LIN {X 0,Y 346.568,Z 1182.724,A -85,B 0,C 180,E1 15595.642,E2 15595.642} C_VEL
LIN {X 0,Y 345.198,Z 1187.452,A -85,B 0,C 180,E1 15592.042,E2 15592.042} C_VEL
LIN {X 0,Y 344.384,Z 1191.307,A -85,B 0,C 180,E1 15588.274,E2 15588.274} C_VEL
LIN {X 0,Y 344.008,Z 1194.426,A -85,B 0,C 180,E1 15583.96,E2 15583.96} C_VEL
LIN {X 0,Y 343.921,Z 1195.912,A -85,B 0,C 180,E1 15579.708,E2 15579.708} C_VEL
LIN {X 0,Y 343.92,Z 1196.098,A -85,B 0,C 180,E1 15576.112,E2 15576.112} C_VEL
LIN {X 0,Y 343.929,Z 1195.312,A -85,B 0,C 180,E1 15572.666,E2 15572.666} C_VEL
LIN {X 0,Y 344.029,Z 1193.649,A -85,B 0,C 180,E1 15569.334,E2 15569.334} C_VEL
LIN {X 0,Y 344.332,Z 1190.938,A -85,B 0,C 180,E1 15565.837,E2 15565.837} C_VEL
LIN {X 0,Y 345.025,Z 1187.235,A -85,B 0,C 180,E1 15562.339,E2 15562.339} C_VEL
LIN {X 0,Y 346.225,Z 1182.52,A -85,B 0,C 180,E1 15558.844,E2 15558.844} C_VEL
LIN {X 0,Y 348.076,Z 1176.766,A -85,B 0,C 180,E1 15555.358,E2 15555.358} C_VEL
LIN {X 0,Y 350.938,Z 1169.245,A -85,B 0,C 180,E1 15551.564,E2 15551.564} C_VEL
LIN {X 0,Y 355.746,Z 1158.187,A -85,B 0,C 180,E1 15547.004,E2 15547.004} C_VEL
LIN {X 0,Y 360.656,Z 1147.928,A -85,B 0,C 180,E1 15543.491,E2 15543.491} C_VEL
LIN {X 0,Y 366.084,Z 1137.114,A -85,B 0,C 180,E1 15540.292,E2 15540.292} C_VEL
LIN {X 0,Y 372.756,Z 1124.27,A -85,B 0,C 180,E1 15537.009,E2 15537.009} C_VEL
LIN {X 0,Y 374.75,Z 1120.524,A -85,B 0,C 180,E1 15536.141,E2 15536.141} C_VEL
LIN {X 0,Y 376.046,Z 1116.491,A -85,B 0,C 180,E1 15535.154,E2 15535.154} C_VEL
LIN {X 0,Y 376.596,Z 1106.617,A -85,B 0,C 180,E1 15532.482,E2 15532.482} C_VEL
LIN {X 0,Y 378.202,Z 1102.238,A -85,B 0,C 180,E1 15531.533,E2 15531.533} C_VEL
LIN {X 0,Y 388.069,Z 1083.778,A -85,B 0,C 180,E1 15528.338,E2 15528.338} C_VEL
LIN {X 0,Y 396.837,Z 1066.652,A -85,B 0,C 180,E1 15525.841,E2 15525.841} C_VEL
LIN {X 0,Y 404.683,Z 1050.76,A -85,B 0,C 180,E1 15523.826,E2 15523.826} C_VEL
LIN {X 0,Y 412.691,Z 1033.763,A -85,B 0,C 180,E1 15521.945,E2 15521.945} C_VEL
LIN {X 0,Y 421.387,Z 1014.239,A -85,B 0,C 180,E1 15520.074,E2 15520.074} C_VEL
LIN {X 0,Y 431.348,Z 989.73,A -85,B 0,C 180,E1 15518.098,E2 15518.098} C_VEL
LIN {X 0,Y 438.671,Z 970.006,A -85,B 0,C 180,E1 15516.758,E2 15516.758} C_VEL
LIN {X 0,Y 445.213,Z 950.609,A -85,B 0,C 180,E1 15515.612,E2 15515.612} C_VEL
LIN {X 0,Y 451.627,Z 929.634,A -85,B 0,C 180,E1 15514.556,E2 15514.556} C_VEL
LIN {X 0,Y 458.617,Z 903.499,A -85,B 0,C 180,E1 15513.46,E2 15513.46} C_VEL
LIN {X 0,Y 464.106,Z 878.646,A -85,B 0,C 180,E1 15512.632,E2 15512.632} C_VEL
LIN {X 0,Y 468.081,Z 857.042,A -85,B 0,C 180,E1 15512.046,E2 15512.046} C_VEL
LIN {X 0,Y 471.395,Z 834.774,A -85,B 0,C 180,E1 15511.57,E2 15511.57} C_VEL
LIN {X 0,Y 474.285,Z 806.407,A -85,B 0,C 180,E1 15511.075,E2 15511.075} C_VEL
LIN {X 0,Y 490.886,Z 583.065,A -85,B 0,C 180,E1 15507.599,E2 15507.599} C_VEL
LIN {X 0,Y 493.757,Z 545.15,A -85,B 0,C 180,E1 15507.001,E2 15507.001} C_VEL
LIN {X 0,Y 486.174,Z 532.933,A -85,B 0,C 180,E1 15504.289,E2 15504.289} C_VEL
LIN {X 0,Y 479.89,Z 523.301,A -85,B 0,C 180,E1 15501.699,E2 15501.699} C_VEL
LIN {X 0,Y 474.547,Z 515.365,A -85,B 0,C 180,E1 15499.126,E2 15499.126} C_VEL
LIN {X 0,Y 471.376,Z 510.666,A -85,B 0,C 180,E1 15497.348,E2 15497.348} C_VEL
LIN {X 0,Y 468.645,Z 506.673,A -85,B 0,C 180,E1 15495.595,E2 15495.595} C_VEL
LIN {X 0,Y 465.572,Z 502.135,A -85,B 0,C 180,E1 15493.222,E2 15493.222} C_VEL
LIN {X 0,Y 462.443,Z 497.864,A -85,B 0,C 180,E1 15489.961,E2 15489.961} C_VEL
LIN {X 0,Y 461.806,Z 496.401,A -85,B 0,C 180,E1 15488.969,E2 15488.969} C_VEL
LIN {X 0,Y 459.954,Z 495.059,A -85,B 0,C 180,E1 15483.739,E2 15483.739} C_VEL
LIN {X 0,Y 461.315,Z 496.134,A -85,B 0,C 180,E1 15478.882,E2 15478.882} C_VEL
LIN {X 0,Y 462.041,Z 496.81,A -85,B 0,C 180,E1 15477.768,E2 15477.768} C_VEL
LIN {X 0,Y 464.243,Z 500.766,A -85,B 0,C 180,E1 15475.058,E2 15475.058} C_VEL
LIN {X 0,Y 465.639,Z 502.27,A -85,B 0,C 180,E1 15473.82,E2 15473.82} C_VEL
LIN {X 0,Y 468.799,Z 506.753,A -85,B 0,C 180,E1 15471.414,E2 15471.414} C_VEL
LIN {X 0,Y 473.05,Z 513.167,A -85,B 0,C 180,E1 15468.787,E2 15468.787} C_VEL
LIN {X 0,Y 477.028,Z 519.005,A -85,B 0,C 180,E1 15466.731,E2 15466.731} C_VEL
LIN {X 0,Y 482.506,Z 527.292,A -85,B 0,C 180,E1 15464.279,E2 15464.279} C_VEL
LIN {X 0,Y 489.139,Z 537.554,A -85,B 0,C 180,E1 15461.713,E2 15461.713} C_VEL
LIN {X 0,Y 493.798,Z 546.364,A -85,B 0,C 180,E1 15460.047,E2 15460.047} C_VEL
LIN {X 0,Y 477.206,Z 767.849,A -85,B 0,C 180,E1 15456.603,E2 15456.603} C_VEL
LIN {X 0,Y 472.628,Z 827.074,A -85,B 0,C 180,E1 15455.658,E2 15455.658} C_VEL
LIN {X 0,Y 468.595,Z 857.357,A -85,B 0,C 180,E1 15455.062,E2 15455.062} C_VEL
LIN {X 0,Y 464.454,Z 880.173,A -85,B 0,C 180,E1 15454.482,E2 15454.482} C_VEL
LIN {X 0,Y 459.845,Z 901.491,A -85,B 0,C 180,E1 15453.806,E2 15453.806} C_VEL
LIN {X 0,Y 454.495,Z 922.797,A -85,B 0,C 180,E1 15452.995,E2 15452.995} C_VEL
LIN {X 0,Y 447.013,Z 948.76,A -85,B 0,C 180,E1 15451.797,E2 15451.797} C_VEL
LIN {X 0,Y 439.383,Z 971.659,A -85,B 0,C 180,E1 15450.506,E2 15450.506} C_VEL
LIN {X 0,Y 432.328,Z 990.947,A -85,B 0,C 180,E1 15449.237,E2 15449.237} C_VEL
LIN {X 0,Y 425.139,Z 1009.177,A -85,B 0,C 180,E1 15447.85,E2 15447.85} C_VEL
LIN {X 0,Y 417.318,Z 1027.631,A -85,B 0,C 180,E1 15446.241,E2 15446.241} C_VEL
LIN {X 0,Y 407.206,Z 1049.934,A -85,B 0,C 180,E1 15443.965,E2 15443.965} C_VEL
LIN {X 0,Y 398.127,Z 1068.568,A -85,B 0,C 180,E1 15441.703,E2 15441.703} C_VEL
LIN {X 0,Y 390.292,Z 1084.053,A -85,B 0,C 180,E1 15439.54,E2 15439.54} C_VEL
LIN {X 0,Y 382.689,Z 1098.648,A -85,B 0,C 180,E1 15437.209,E2 15437.209} C_VEL
LIN {X 0,Y 374.954,Z 1113.254,A -85,B 0,C 180,E1 15434.533,E2 15434.533} C_VEL
LIN {X 0,Y 365.691,Z 1130.554,A -85,B 0,C 180,E1 15430.803,E2 15430.803} C_VEL
LIN {X 0,Y 358.982,Z 1143.123,A -85,B 0,C 180,E1 15427.587,E2 15427.587} C_VEL
LIN {X 0,Y 353.255,Z 1154.282,A -85,B 0,C 180,E1 15424.281,E2 15424.281} C_VEL
LIN {X 0,Y 348.218,Z 1164.594,A -85,B 0,C 180,E1 15420.737,E2 15420.737} C_VEL
LIN {X 0,Y 343.21,Z 1175.867,A -85,B 0,C 180,E1 15416.097,E2 15416.097} C_VEL
LIN {X 0,Y 340.131,Z 1183.761,A -85,B 0,C 180,E1 15412.103,E2 15412.103} C_VEL
LIN {X 0,Y 338.181,Z 1189.769,A -85,B 0,C 180,E1 15408.442,E2 15408.442} C_VEL
LIN {X 0,Y 336.997,Z 1194.445,A -85,B 0,C 180,E1 15404.959,E2 15404.959} C_VEL
LIN {X 0,Y 336.305,Z 1198.13,A -85,B 0,C 180,E1 15401.49,E2 15401.49} C_VEL
LIN {X 0,Y 336.02,Z 1200.852,A -85,B 0,C 180,E1 15398.039,E2 15398.039} C_VEL
LIN {X 0,Y 335.924,Z 1202.564,A -85,B 0,C 180,E1 15394.781,E2 15394.781} C_VEL
LIN {X 0,Y 335.915,Z 1203.44,A -85,B 0,C 180,E1 15391.535,E2 15391.535} C_VEL
LIN {X 0,Y 335.913,Z 1203.49,A -85,B 0,C 180,E1 15388.294,E2 15388.294} C_VEL
LIN {X 0,Y 335.926,Z 1202.719,A -85,B 0,C 180,E1 15385.048,E2 15385.048} C_VEL
LIN {X 0,Y 336.037,Z 1201.013,A -85,B 0,C 180,E1 15381.617,E2 15381.617} C_VEL
LIN {X 0,Y 336.388,Z 1198.232,A -85,B 0,C 180,E1 15377.991,E2 15377.991} C_VEL
LIN {X 0,Y 337.167,Z 1194.642,A -85,B 0,C 180,E1 15374.521,E2 15374.521} C_VEL
LIN {X 0,Y 338.55,Z 1189.852,A -85,B 0,C 180,E1 15370.863,E2 15370.863} C_VEL
LIN {X 0,Y 340.701,Z 1183.995,A -85,B 0,C 180,E1 15367.208,E2 15367.208} C_VEL
LIN {X 0,Y 343.862,Z 1176.688,A -85,B 0,C 180,E1 15363.398,E2 15363.398} C_VEL
LIN {X 0,Y 349.185,Z 1166.017,A -85,B 0,C 180,E1 15358.783,E2 15358.783} C_VEL
LIN {X 0,Y 355.02,Z 1155.183,A -85,B 0,C 180,E1 15354.933,E2 15354.933} C_VEL
LIN {X 0,Y 361.14,Z 1144.496,A -85,B 0,C 180,E1 15351.672,E2 15351.672} C_VEL
LIN {X 0,Y 368.243,Z 1132.499,A -85,B 0,C 180,E1 15348.508,E2 15348.508} C_VEL
LIN {X 0,Y 377.138,Z 1117.696,A -85,B 0,C 180,E1 15345.154,E2 15345.154} C_VEL
LIN {X 0,Y 387.584,Z 1099.925,A -85,B 0,C 180,E1 15341.795,E2 15341.795} C_VEL
LIN {X 0,Y 396.6,Z 1084.321,A -85,B 0,C 180,E1 15339.288,E2 15339.288} C_VEL
LIN {X 0,Y 405.359,Z 1068.713,A -85,B 0,C 180,E1 15337.118,E2 15337.118} C_VEL
LIN {X 0,Y 415.508,Z 1049.873,A -85,B 0,C 180,E1 15334.859,E2 15334.859} C_VEL
LIN {X 0,Y 426.712,Z 1027.473,A -85,B 0,C 180,E1 15332.612,E2 15332.612} C_VEL
LIN {X 0,Y 435.312,Z 1009.07,A -85,B 0,C 180,E1 15331.048,E2 15331.048} C_VEL
LIN {X 0,Y 443.198,Z 990.925,A -85,B 0,C 180,E1 15329.708,E2 15329.708} C_VEL
LIN {X 0,Y 450.955,Z 971.577,A -85,B 0,C 180,E1 15328.471,E2 15328.471} C_VEL
LIN {X 0,Y 459.654,Z 947.749,A -85,B 0,C 180,E1 15327.182,E2 15327.182} C_VEL
LIN {X 0,Y 467.531,Z 922.667,A -85,B 0,C 180,E1 15326.077,E2 15326.077} C_VEL
LIN {X 0,Y 473.352,Z 901.443,A -85,B 0,C 180,E1 15325.303,E2 15325.303} C_VEL
LIN {X 0,Y 478.364,Z 880.268,A -85,B 0,C 180,E1 15324.665,E2 15324.665} C_VEL
LIN {X 0,Y 482.642,Z 858.736,A -85,B 0,C 180,E1 15324.14,E2 15324.14} C_VEL
LIN {X 0,Y 486.899,Z 831.241,A -85,B 0,C 180,E1 15323.605,E2 15323.605} C_VEL
LIN {X 0,Y 491.021,Z 786.034,A -85,B 0,C 180,E1 15322.885,E2 15322.885} C_VEL
LIN {X 0,Y 509.816,Z 566.031,A -85,B 0,C 180,E1 15319.504,E2 15319.504} C_VEL
LIN {X 0,Y 510.711,Z 555.321,A -85,B 0,C 180,E1 15319.322,E2 15319.322} C_VEL
LIN {X 0,Y 506.863,Z 548.626,A -85,B 0,C 180,E1 15317.389,E2 15317.389} C_VEL
LIN {X 0,Y 503.453,Z 543.319,A -85,B 0,C 180,E1 15315.434,E2 15315.434} C_VEL
LIN {X 0,Y 501.187,Z 539.639,A -85,B 0,C 180,E1 15313.91,E2 15313.91} C_VEL
LIN {X 0,Y 498.572,Z 535.499,A -85,B 0,C 180,E1 15311.804,E2 15311.804} C_VEL
LIN {X 0,Y 495.748,Z 530.771,A -85,B 0,C 180,E1 15308.584,E2 15308.584} C_VEL
LIN {X 0,Y 493.92,Z 528.892,A -85,B 0,C 180,E1 15303.831,E2 15303.831} C_VEL
LIN {X 0,Y 494.308,Z 529.49,A -85,B 0,C 180,E1 15300.927,E2 15300.927} C_VEL
LIN {X 0,Y 495.953,Z 531.071,A -85,B 0,C 180,E1 15297.92,E2 15297.92} C_VEL
LIN {X 0,Y 498.766,Z 535.705,A -85,B 0,C 180,E1 15294.824,E2 15294.824} C_VEL
LIN {X 0,Y 502.313,Z 541.374,A -85,B 0,C 180,E1 15292.105,E2 15292.105} C_VEL
LIN {X 0,Y 505.598,Z 546.687,A -85,B 0,C 180,E1 15290.093,E2 15290.093} C_VEL
LIN {X 0,Y 509.935,Z 553.595,A -85,B 0,C 180,E1 15287.86,E2 15287.86} C_VEL
LIN {X 0,Y 510.673,Z 555.182,A -85,B 0,C 180,E1 15287.494,E2 15287.494} C_VEL
LIN {X 0,Y 492.196,Z 770.494,A -85,B 0,C 180,E1 15284.188,E2 15284.188} C_VEL
LIN {X 0,Y 487.454,Z 823.866,A -85,B 0,C 180,E1 15283.347,E2 15283.347} C_VEL
LIN {X 0,Y 483.136,Z 853.307,A -85,B 0,C 180,E1 15282.782,E2 15282.782} C_VEL
LIN {X 0,Y 478.728,Z 875.802,A -85,B 0,C 180,E1 15282.224,E2 15282.224} C_VEL
LIN {X 0,Y 473.908,Z 896.408,A -85,B 0,C 180,E1 15281.592,E2 15281.592} C_VEL
LIN {X 0,Y 468.336,Z 916.956,A -85,B 0,C 180,E1 15280.837,E2 15280.837} C_VEL
LIN {X 0,Y 461.23,Z 939.95,A -85,B 0,C 180,E1 15279.827,E2 15279.827} C_VEL
LIN {X 0,Y 452.08,Z 965.513,A -85,B 0,C 180,E1 15278.46,E2 15278.46} C_VEL
LIN {X 0,Y 444.164,Z 985.323,A -85,B 0,C 180,E1 15277.194,E2 15277.194} C_VEL
LIN {X 0,Y 436.186,Z 1003.729,A -85,B 0,C 180,E1 15275.828,E2 15275.828} C_VEL
LIN {X 0,Y 427.778,Z 1021.716,A -85,B 0,C 180,E1 15274.295,E2 15274.295} C_VEL
LIN {X 0,Y 417.178,Z 1043.001,A -85,B 0,C 180,E1 15272.176,E2 15272.176} C_VEL
LIN {X 0,Y 406.533,Z 1062.656,A -85,B 0,C 180,E1 15269.826,E2 15269.826} C_VEL
LIN {X 0,Y 397.526,Z 1078.589,A -85,B 0,C 180,E1 15267.605,E2 15267.605} C_VEL
LIN {X 0,Y 389.142,Z 1092.928,A -85,B 0,C 180,E1 15265.306,E2 15265.306} C_VEL
LIN {X 0,Y 380.303,Z 1107.754,A -85,B 0,C 180,E1 15262.56,E2 15262.56} C_VEL
LIN {X 0,Y 369.726,Z 1125.201,A -85,B 0,C 180,E1 15258.709,E2 15258.709} C_VEL
LIN {X 0,Y 362.319,Z 1137.42,A -85,B 0,C 180,E1 15255.495,E2 15255.495} C_VEL
LIN {X 0,Y 356.234,Z 1147.753,A -85,B 0,C 180,E1 15252.347,E2 15252.347} C_VEL
LIN {X 0,Y 350.658,Z 1157.649,A -85,B 0,C 180,E1 15248.851,E2 15248.851} C_VEL
LIN {X 0,Y 345.045,Z 1168.446,A -85,B 0,C 180,E1 15244.321,E2 15244.321} C_VEL
LIN {X 0,Y 341.235,Z 1176.607,A -85,B 0,C 180,E1 15240.069,E2 15240.069} C_VEL
LIN {X 0,Y 338.869,Z 1182.639,A -85,B 0,C 180,E1 15236.269,E2 15236.269} C_VEL
LIN {X 0,Y 337.392,Z 1187.309,A -85,B 0,C 180,E1 15232.659,E2 15232.659} C_VEL
LIN {X 0,Y 336.513,Z 1190.964,A -85,B 0,C 180,E1 15229.077,E2 15229.077} C_VEL
LIN {X 0,Y 336.103,Z 1193.64,A -85,B 0,C 180,E1 15225.53,E2 15225.53} C_VEL
LIN {X 0,Y 335.947,Z 1195.365,A -85,B 0,C 180,E1 15222.025,E2 15222.025} C_VEL
LIN {X 0,Y 335.919,Z 1196.141,A -85,B 0,C 180,E1 15218.731,E2 15218.731} C_VEL
LIN {X 0,Y 335.92,Z 1196.095,A -85,B 0,C 180,E1 15215.466,E2 15215.466} C_VEL
LIN {X 0,Y 335.935,Z 1195.243,A -85,B 0,C 180,E1 15212.217,E2 15212.217} C_VEL
LIN {X 0,Y 336.05,Z 1193.589,A -85,B 0,C 180,E1 15208.977,E2 15208.977} C_VEL
LIN {X 0,Y 336.367,Z 1190.976,A -85,B 0,C 180,E1 15205.567,E2 15205.567} C_VEL
LIN {X 0,Y 337.119,Z 1187.259,A -85,B 0,C 180,E1 15201.987,E2 15201.987} C_VEL
LIN {X 0,Y 338.413,Z 1182.528,A -85,B 0,C 180,E1 15198.41,E2 15198.41} C_VEL
LIN {X 0,Y 340.488,Z 1176.462,A -85,B 0,C 180,E1 15194.675,E2 15194.675} C_VEL
LIN {X 0,Y 344.061,Z 1167.84,A -85,B 0,C 180,E1 15190.3,E2 15190.3} C_VEL
LIN {X 0,Y 348.939,Z 1157.229,A -85,B 0,C 180,E1 15185.991,E2 15185.991} C_VEL
LIN {X 0,Y 353.92,Z 1147.346,A -85,B 0,C 180,E1 15182.581,E2 15182.581} C_VEL
LIN {X 0,Y 359.513,Z 1136.701,A -85,B 0,C 180,E1 15179.406,E2 15179.406} C_VEL
LIN {X 0,Y 367.403,Z 1122.28,A -85,B 0,C 180,E1 15175.713,E2 15175.713} C_VEL
LIN {X 0,Y 376.061,Z 1106.21,A -85,B 0,C 180,E1 15172.301,E2 15172.301} C_VEL
LIN {X 0,Y 378.202,Z 1102.238,A -85,B 0,C 180,E1 15171.533,E2 15171.533} C_VEL
LIN {X 0,Y 379.88,Z 1097.862,A -85,B 0,C 180,E1 15170.598,E2 15170.598} C_VEL
LIN {X 0,Y 381.583,Z 1086.344,A -85,B 0,C 180,E1 15167.924,E2 15167.924} C_VEL
LIN {X 0,Y 383.266,Z 1082.167,A -85,B 0,C 180,E1 15167.189,E2 15167.189} C_VEL
LIN {X 0,Y 391.871,Z 1065.862,A -85,B 0,C 180,E1 15164.821,E2 15164.821} C_VEL
LIN {X 0,Y 399.975,Z 1049.884,A -85,B 0,C 180,E1 15162.803,E2 15162.803} C_VEL
LIN {X 0,Y 408.506,Z 1032.191,A -85,B 0,C 180,E1 15160.861,E2 15160.861} C_VEL
LIN {X 0,Y 418.945,Z 1009.024,A -85,B 0,C 180,E1 15158.701,E2 15158.701} C_VEL
LIN {X 0,Y 427.583,Z 987.921,A -85,B 0,C 180,E1 15157.053,E2 15157.053} C_VEL
LIN {X 0,Y 434.914,Z 968.488,A -85,B 0,C 180,E1 15155.754,E2 15155.754} C_VEL
LIN {X 0,Y 441.595,Z 948.987,A -85,B 0,C 180,E1 15154.622,E2 15154.622} C_VEL
LIN {X 0,Y 449.208,Z 924.376,A -85,B 0,C 180,E1 15153.417,E2 15153.417} C_VEL
LIN {X 0,Y 455.898,Z 898.52,A -85,B 0,C 180,E1 15152.396,E2 15152.396} C_VEL
LIN {X 0,Y 460.648,Z 877.08,A -85,B 0,C 180,E1 15151.703,E2 15151.703} C_VEL
LIN {X 0,Y 464.647,Z 855.505,A -85,B 0,C 180,E1 15151.133,E2 15151.133} C_VEL
LIN {X 0,Y 468.365,Z 830.302,A -85,B 0,C 180,E1 15150.611,E2 15150.611} C_VEL
LIN {X 0,Y 471.673,Z 793.271,A -85,B 0,C 180,E1 15149.998,E2 15149.998} C_VEL
LIN {X 0,Y 488.775,Z 569.761,A -85,B 0,C 180,E1 15146.528,E2 15146.528} C_VEL
LIN {X 0,Y 490.239,Z 550.028,A -85,B 0,C 180,E1 15146.198,E2 15146.198} C_VEL
LIN {X 0,Y 482.382,Z 537.211,A -85,B 0,C 180,E1 15143.226,E2 15143.226} C_VEL
LIN {X 0,Y 476.274,Z 527.795,A -85,B 0,C 180,E1 15140.524,E2 15140.524} C_VEL
LIN {X 0,Y 470.602,Z 519.114,A -85,B 0,C 180,E1 15137.496,E2 15137.496} C_VEL
LIN {X 0,Y 467.144,Z 514.202,A -85,B 0,C 180,E1 15135.264,E2 15135.264} C_VEL
LIN {X 0,Y 463.967,Z 509.456,A -85,B 0,C 180,E1 15132.699,E2 15132.699} C_VEL
LIN {X 0,Y 461.331,Z 505.676,A -85,B 0,C 180,E1 15129.796,E2 15129.796} C_VEL
LIN {X 0,Y 460.751,Z 504.308,A -85,B 0,C 180,E1 15128.863,E2 15128.863} C_VEL
LIN {X 0,Y 458.978,Z 502.999,A -85,B 0,C 180,E1 15123.747,E2 15123.747} C_VEL
LIN {X 0,Y 460.337,Z 504.081,A -85,B 0,C 180,E1 15118.88,E2 15118.88} C_VEL
LIN {X 0,Y 460.969,Z 504.715,A -85,B 0,C 180,E1 15117.887,E2 15117.887} C_VEL
LIN {X 0,Y 463.132,Z 508.635,A -85,B 0,C 180,E1 15115.17,E2 15115.17} C_VEL
LIN {X 0,Y 464.481,Z 510.181,A -85,B 0,C 180,E1 15113.945,E2 15113.945} C_VEL
LIN {X 0,Y 468.144,Z 515.561,A -85,B 0,C 180,E1 15111.154,E2 15111.154} C_VEL
LIN {X 0,Y 471.623,Z 520.862,A -85,B 0,C 180,E1 15109,E2 15109} C_VEL
LIN {X 0,Y 475.54,Z 526.709,A -85,B 0,C 180,E1 15106.936,E2 15106.936} C_VEL
LIN {X 0,Y 481.28,Z 535.588,A -85,B 0,C 180,E1 15104.331,E2 15104.331} C_VEL
LIN {X 0,Y 487.263,Z 545.065,A -85,B 0,C 180,E1 15101.98,E2 15101.98} C_VEL
LIN {X 0,Y 490.333,Z 551.144,A -85,B 0,C 180,E1 15100.837,E2 15100.837} C_VEL
LIN {X 0,Y 473.346,Z 772.468,A -85,B 0,C 180,E1 15097.4,E2 15097.4} C_VEL
LIN {X 0,Y 468.94,Z 827.656,A -85,B 0,C 180,E1 15096.519,E2 15096.519} C_VEL
LIN {X 0,Y 464.851,Z 857.543,A -85,B 0,C 180,E1 15095.932,E2 15095.932} C_VEL
LIN {X 0,Y 460.661,Z 880.186,A -85,B 0,C 180,E1 15095.359,E2 15095.359} C_VEL
LIN {X 0,Y 456.1,Z 900.89,A -85,B 0,C 180,E1 15094.711,E2 15094.711} C_VEL
LIN {X 0,Y 450.629,Z 922.307,A -85,B 0,C 180,E1 15093.904,E2 15093.904} C_VEL
LIN {X 0,Y 443.158,Z 947.845,A -85,B 0,C 180,E1 15092.74,E2 15092.74} C_VEL
LIN {X 0,Y 435.014,Z 971.75,A -85,B 0,C 180,E1 15091.403,E2 15091.403} C_VEL
LIN {X 0,Y 427.768,Z 991.112,A -85,B 0,C 180,E1 15090.131,E2 15090.131} C_VEL
LIN {X 0,Y 420.123,Z 1009.995,A -85,B 0,C 180,E1 15088.692,E2 15088.692} C_VEL
LIN {X 0,Y 411.515,Z 1029.732,A -85,B 0,C 180,E1 15086.955,E2 15086.955} C_VEL
LIN {X 0,Y 400.691,Z 1052.623,A -85,B 0,C 180,E1 15084.56,E2 15084.56} C_VEL
LIN {X 0,Y 392.15,Z 1069.632,A -85,B 0,C 180,E1 15082.462,E2 15082.462} C_VEL
LIN {X 0,Y 384.07,Z 1085.085,A -85,B 0,C 180,E1 15080.272,E2 15080.272} C_VEL
LIN {X 0,Y 375.661,Z 1100.713,A -85,B 0,C 180,E1 15077.725,E2 15077.725} C_VEL
LIN {X 0,Y 365.605,Z 1118.951,A -85,B 0,C 180,E1 15074.217,E2 15074.217} C_VEL
LIN {X 0,Y 357.76,Z 1132.963,A -85,B 0,C 180,E1 15071.008,E2 15071.008} C_VEL
LIN {X 0,Y 351.354,Z 1144.58,A -85,B 0,C 180,E1 15067.928,E2 15067.928} C_VEL
LIN {X 0,Y 345.498,Z 1155.583,A -85,B 0,C 180,E1 15064.556,E2 15064.556} C_VEL
LIN {X 0,Y 339.274,Z 1167.956,A -85,B 0,C 180,E1 15060.066,E2 15060.066} C_VEL
LIN {X 0,Y 335.072,Z 1177.098,A -85,B 0,C 180,E1 15056.018,E2 15056.018} C_VEL
LIN {X 0,Y 332.214,Z 1184.19,A -85,B 0,C 180,E1 15052.285,E2 15052.285} C_VEL
LIN {X 0,Y 330.208,Z 1190.116,A -85,B 0,C 180,E1 15048.538,E2 15048.538} C_VEL
LIN {X 0,Y 328.903,Z 1195.132,A -85,B 0,C 180,E1 15044.615,E2 15044.615} C_VEL
LIN {X 0,Y 328.15,Z 1199.574,A -85,B 0,C 180,E1 15040.002,E2 15040.002} C_VEL
LIN {X 0,Y 327.942,Z 1202.111,A -85,B 0,C 180,E1 15035.774,E2 15035.774} C_VEL
LIN {X 0,Y 327.913,Z 1203.278,A -85,B 0,C 180,E1 15032.097,E2 15032.097} C_VEL
LIN {X 0,Y 327.916,Z 1203.456,A -85,B 0,C 180,E1 15028.602,E2 15028.602} C_VEL
LIN {X 0,Y 327.928,Z 1202.65,A -85,B 0,C 180,E1 15024.927,E2 15024.927} C_VEL
LIN {X 0,Y 328.05,Z 1200.958,A -85,B 0,C 180,E1 15021.411,E2 15021.411} C_VEL
LIN {X 0,Y 328.437,Z 1198.193,A -85,B 0,C 180,E1 15017.696,E2 15017.696} C_VEL
LIN {X 0,Y 329.332,Z 1194.41,A -85,B 0,C 180,E1 15013.962,E2 15013.962} C_VEL
LIN {X 0,Y 330.853,Z 1189.59,A -85,B 0,C 180,E1 15010.216,E2 15010.216} C_VEL
LIN {X 0,Y 333.193,Z 1183.704,A -85,B 0,C 180,E1 15006.477,E2 15006.477} C_VEL
LIN {X 0,Y 336.785,Z 1176.014,A -85,B 0,C 180,E1 15002.41,E2 15002.41} C_VEL
LIN {X 0,Y 342.779,Z 1164.723,A -85,B 0,C 180,E1 14997.54,E2 14997.54} C_VEL
LIN {X 0,Y 348.791,Z 1154.258,A -85,B 0,C 180,E1 14993.806,E2 14993.806} C_VEL
LIN {X 0,Y 355.32,Z 1143.481,A -85,B 0,C 180,E1 14990.509,E2 14990.509} C_VEL
LIN {X 0,Y 363.201,Z 1130.763,A -85,B 0,C 180,E1 14987.159,E2 14987.159} C_VEL
LIN {X 0,Y 373.952,Z 1113.446,A -85,B 0,C 180,E1 14983.343,E2 14983.343} C_VEL
LIN {X 0,Y 383.086,Z 1098.498,A -85,B 0,C 180,E1 14980.579,E2 14980.579} C_VEL
LIN {X 0,Y 391.943,Z 1083.684,A -85,B 0,C 180,E1 14978.213,E2 14978.213} C_VEL
LIN {X 0,Y 401.418,Z 1067.305,A -85,B 0,C 180,E1 14975.952,E2 14975.952} C_VEL
LIN {X 0,Y 413.3,Z 1045.658,A -85,B 0,C 180,E1 14973.423,E2 14973.423} C_VEL
LIN {X 0,Y 423.336,Z 1025.935,A -85,B 0,C 180,E1 14971.501,E2 14971.501} C_VEL
LIN {X 0,Y 432.189,Z 1007.376,A -85,B 0,C 180,E1 14969.951,E2 14969.951} C_VEL
LIN {X 0,Y 440.294,Z 989.092,A -85,B 0,C 180,E1 14968.632,E2 14968.632} C_VEL
LIN {X 0,Y 449.321,Z 966.871,A -85,B 0,C 180,E1 14967.253,E2 14967.253} C_VEL
LIN {X 0,Y 458.251,Z 941.934,A -85,B 0,C 180,E1 14965.981,E2 14965.981} C_VEL
LIN {X 0,Y 464.824,Z 921.12,A -85,B 0,C 180,E1 14965.097,E2 14965.097} C_VEL
LIN {X 0,Y 470.581,Z 900.399,A -85,B 0,C 180,E1 14964.36,E2 14964.36} C_VEL
LIN {X 0,Y 475.668,Z 879.161,A -85,B 0,C 180,E1 14963.734,E2 14963.734} C_VEL
LIN {X 0,Y 480.278,Z 856.07,A -85,B 0,C 180,E1 14963.186,E2 14963.186} C_VEL
LIN {X 0,Y 484.648,Z 826.198,A -85,B 0,C 180,E1 14962.633,E2 14962.633} C_VEL
LIN {X 0,Y 490.49,Z 760.806,A -85,B 0,C 180,E1 14961.611,E2 14961.611} C_VEL
LIN {X 0,Y 508.048,Z 560.807,A -85,B 0,C 180,E1 14958.548,E2 14958.548} C_VEL
LIN {X 0,Y 504.157,Z 554.3,A -85,B 0,C 180,E1 14956.476,E2 14956.476} C_VEL
LIN {X 0,Y 500.136,Z 547.649,A -85,B 0,C 180,E1 14953.881,E2 14953.881} C_VEL
LIN {X 0,Y 497.344,Z 543.242,A -85,B 0,C 180,E1 14951.598,E2 14951.598} C_VEL
LIN {X 0,Y 494.693,Z 538.674,A -85,B 0,C 180,E1 14948.485,E2 14948.485} C_VEL
LIN {X 0,Y 492.938,Z 536.815,A -85,B 0,C 180,E1 14943.722,E2 14943.722} C_VEL
LIN {X 0,Y 493.368,Z 537.484,A -85,B 0,C 180,E1 14940.813,E2 14940.813} C_VEL
LIN {X 0,Y 494.919,Z 539.073,A -85,B 0,C 180,E1 14937.974,E2 14937.974} C_VEL
LIN {X 0,Y 498.083,Z 544.421,A -85,B 0,C 180,E1 14934.528,E2 14934.528} C_VEL
LIN {X 0,Y 501.058,Z 549.201,A -85,B 0,C 180,E1 14932.259,E2 14932.259} C_VEL
LIN {X 0,Y 504.293,Z 554.533,A -85,B 0,C 180,E1 14930.24,E2 14930.24} C_VEL
LIN {X 0,Y 507.99,Z 560.589,A -85,B 0,C 180,E1 14928.282,E2 14928.282} C_VEL
LIN {X 0,Y 488.97,Z 777.287,A -85,B 0,C 180,E1 14924.97,E2 14924.97} C_VEL
LIN {X 0,Y 484.525,Z 825.48,A -85,B 0,C 180,E1 14924.21,E2 14924.21} C_VEL
LIN {X 0,Y 480.195,Z 853.913,A -85,B 0,C 180,E1 14923.664,E2 14923.664} C_VEL
LIN {X 0,Y 475.748,Z 876.139,A -85,B 0,C 180,E1 14923.118,E2 14923.118} C_VEL
LIN {X 0,Y 470.762,Z 897.009,A -85,B 0,C 180,E1 14922.484,E2 14922.484} C_VEL
LIN {X 0,Y 464.911,Z 918.08,A -85,B 0,C 180,E1 14921.714,E2 14921.714} C_VEL
LIN {X 0,Y 456.877,Z 943.312,A -85,B 0,C 180,E1 14920.6,E2 14920.6} C_VEL
LIN {X 0,Y 448.133,Z 966.801,A -85,B 0,C 180,E1 14919.331,E2 14919.331} C_VEL
LIN {X 0,Y 440.213,Z 986.124,A -85,B 0,C 180,E1 14918.099,E2 14918.099} C_VEL
LIN {X 0,Y 432.403,Z 1003.693,A -85,B 0,C 180,E1 14916.802,E2 14916.802} C_VEL
LIN {X 0,Y 423.777,Z 1021.68,A -85,B 0,C 180,E1 14915.28,E2 14915.28} C_VEL
LIN {X 0,Y 412.889,Z 1042.975,A -85,B 0,C 180,E1 14913.172,E2 14913.172} C_VEL
LIN {X 0,Y 401.853,Z 1062.765,A -85,B 0,C 180,E1 14910.811,E2 14910.811} C_VEL
LIN {X 0,Y 392.514,Z 1078.773,A -85,B 0,C 180,E1 14908.578,E2 14908.578} C_VEL
LIN {X 0,Y 383.374,Z 1093.879,A -85,B 0,C 180,E1 14906.139,E2 14906.139} C_VEL
LIN {X 0,Y 372.766,Z 1111.1,A -85,B 0,C 180,E1 14902.877,E2 14902.877} C_VEL
LIN {X 0,Y 363.202,Z 1126.082,A -85,B 0,C 180,E1 14899.446,E2 14899.446} C_VEL
LIN {X 0,Y 355.635,Z 1138.049,A -85,B 0,C 180,E1 14896.239,E2 14896.239} C_VEL
LIN {X 0,Y 349.146,Z 1148.56,A -85,B 0,C 180,E1 14892.966,E2 14892.966} C_VEL
LIN {X 0,Y 342.572,Z 1159.786,A -85,B 0,C 180,E1 14888.867,E2 14888.867} C_VEL
LIN {X 0,Y 336.981,Z 1169.949,A -85,B 0,C 180,E1 14884.315,E2 14884.315} C_VEL
LIN {X 0,Y 333.494,Z 1177.111,A -85,B 0,C 180,E1 14880.443,E2 14880.443} C_VEL
LIN {X 0,Y 331.103,Z 1182.816,A -85,B 0,C 180,E1 14876.74,E2 14876.74} C_VEL
LIN {X 0,Y 329.523,Z 1187.468,A -85,B 0,C 180,E1 14873.043,E2 14873.043} C_VEL
LIN {X 0,Y 328.571,Z 1191.107,A -85,B 0,C 180,E1 14869.371,E2 14869.371} C_VEL
LIN {X 0,Y 328.113,Z 1193.828,A -85,B 0,C 180,E1 14865.638,E2 14865.638} C_VEL
LIN {X 0,Y 327.946,Z 1195.544,A -85,B 0,C 180,E1 14861.965,E2 14861.965} C_VEL
LIN {X 0,Y 327.916,Z 1196.303,A -85,B 0,C 180,E1 14858.239,E2 14858.239} C_VEL
LIN {X 0,Y 327.917,Z 1196.017,A -85,B 0,C 180,E1 14854.197,E2 14854.197} C_VEL
LIN {X 0,Y 328.017,Z 1194.313,A -85,B 0,C 180,E1 14849.825,E2 14849.825} C_VEL
LIN {X 0,Y 328.34,Z 1191.483,A -85,B 0,C 180,E1 14845.809,E2 14845.809} C_VEL
LIN {X 0,Y 329.125,Z 1187.684,A -85,B 0,C 180,E1 14841.967,E2 14841.967} C_VEL
LIN {X 0,Y 330.452,Z 1183.031,A -85,B 0,C 180,E1 14838.304,E2 14838.304} C_VEL
LIN {X 0,Y 332.478,Z 1177.339,A -85,B 0,C 180,E1 14834.654,E2 14834.654} C_VEL
LIN {X 0,Y 335.465,Z 1170.224,A -85,B 0,C 180,E1 14830.861,E2 14830.861} C_VEL
LIN {X 0,Y 340.242,Z 1160.291,A -85,B 0,C 180,E1 14826.443,E2 14826.443} C_VEL
LIN {X 0,Y 346.205,Z 1148.76,A -85,B 0,C 180,E1 14822.291,E2 14822.291} C_VEL
LIN {X 0,Y 351.929,Z 1138.264,A -85,B 0,C 180,E1 14819.054,E2 14819.054} C_VEL
LIN {X 0,Y 358.542,Z 1126.473,A -85,B 0,C 180,E1 14815.908,E2 14815.908} C_VEL
LIN {X 0,Y 367.399,Z 1110.984,A -85,B 0,C 180,E1 14812.37,E2 14812.37} C_VEL
LIN {X 0,Y 376.873,Z 1093.857,A -85,B 0,C 180,E1 14809.125,E2 14809.125} C_VEL
LIN {X 0,Y 383.266,Z 1082.167,A -85,B 0,C 180,E1 14807.189,E2 14807.189} C_VEL
LIN {X 0,Y 385.174,Z 1077.354,A -85,B 0,C 180,E1 14806.337,E2 14806.337} C_VEL
LIN {X 0,Y 387.469,Z 1065.512,A -85,B 0,C 180,E1 14803.947,E2 14803.947} C_VEL
LIN {X 0,Y 389.584,Z 1060.327,A -85,B 0,C 180,E1 14803.143,E2 14803.143} C_VEL
LIN {X 0,Y 400.455,Z 1038.903,A -85,B 0,C 180,E1 14800.622,E2 14800.622} C_VEL
LIN {X 0,Y 409.201,Z 1020.505,A -85,B 0,C 180,E1 14798.789,E2 14798.789} C_VEL
LIN {X 0,Y 417.074,Z 1002.797,A -85,B 0,C 180,E1 14797.259,E2 14797.259} C_VEL
LIN {X 0,Y 424.873,Z 983.853,A -85,B 0,C 180,E1 14795.834,E2 14795.834} C_VEL
LIN {X 0,Y 433.913,Z 959.888,A -85,B 0,C 180,E1 14794.302,E2 14794.302} C_VEL
LIN {X 0,Y 441.827,Z 935.755,A -85,B 0,C 180,E1 14793.036,E2 14793.036} C_VEL
LIN {X 0,Y 447.808,Z 915.253,A -85,B 0,C 180,E1 14792.131,E2 14792.131} C_VEL
LIN {X 0,Y 452.899,Z 895.386,A -85,B 0,C 180,E1 14791.387,E2 14791.387} C_VEL
LIN {X 0,Y 457.773,Z 873.268,A -85,B 0,C 180,E1 14790.698,E2 14790.698} C_VEL
LIN {X 0,Y 462.739,Z 845.528,A -85,B 0,C 180,E1 14790.021,E2 14790.021} C_VEL
LIN {X 0,Y 465.963,Z 819.816,A -85,B 0,C 180,E1 14789.544,E2 14789.544} C_VEL
LIN {X 0,Y 479.845,Z 643.836,A -85,B 0,C 180,E1 14786.797,E2 14786.797} C_VEL
LIN {X 0,Y 486.897,Z 555.177,A -85,B 0,C 180,E1 14785.417,E2 14785.417} C_VEL
LIN {X 0,Y 480.281,Z 544.19,A -85,B 0,C 180,E1 14782.815,E2 14782.815} C_VEL
LIN {X 0,Y 474.447,Z 535.016,A -85,B 0,C 180,E1 14780.156,E2 14780.156} C_VEL
LIN {X 0,Y 469.124,Z 526.694,A -85,B 0,C 180,E1 14777.233,E2 14777.233} C_VEL
LIN {X 0,Y 465.831,Z 521.916,A -85,B 0,C 180,E1 14775.054,E2 14775.054} C_VEL
LIN {X 0,Y 462.723,Z 517.219,A -85,B 0,C 180,E1 14772.479,E2 14772.479} C_VEL
LIN {X 0,Y 460.184,Z 513.385,A -85,B 0,C 180,E1 14769.568,E2 14769.568} C_VEL
LIN {X 0,Y 459.615,Z 512.169,A -85,B 0,C 180,E1 14768.633,E2 14768.633} C_VEL
LIN {X 0,Y 458,Z 510.937,A -85,B 0,C 180,E1 14763.63,E2 14763.63} C_VEL
LIN {X 0,Y 459.433,Z 512.077,A -85,B 0,C 180,E1 14758.753,E2 14758.753} C_VEL
LIN {X 0,Y 459.935,Z 512.727,A -85,B 0,C 180,E1 14757.944,E2 14757.944} C_VEL
LIN {X 0,Y 462.148,Z 516.641,A -85,B 0,C 180,E1 14755.16,E2 14755.16} C_VEL
LIN {X 0,Y 463.279,Z 517.99,A -85,B 0,C 180,E1 14754.116,E2 14754.116} C_VEL
LIN {X 0,Y 466.875,Z 523.394,A -85,B 0,C 180,E1 14751.316,E2 14751.316} C_VEL
LIN {X 0,Y 470.202,Z 528.555,A -85,B 0,C 180,E1 14749.214,E2 14749.214} C_VEL
LIN {X 0,Y 474.056,Z 534.41,A -85,B 0,C 180,E1 14747.143,E2 14747.143} C_VEL
LIN {X 0,Y 479.851,Z 543.55,A -85,B 0,C 180,E1 14744.469,E2 14744.469} C_VEL
LIN {X 0,Y 485.469,Z 552.716,A -85,B 0,C 180,E1 14742.221,E2 14742.221} C_VEL
LIN {X 0,Y 486.972,Z 555.805,A -85,B 0,C 180,E1 14741.64,E2 14741.64} C_VEL
LIN {X 0,Y 469.631,Z 776.379,A -85,B 0,C 180,E1 14738.222,E2 14738.222} C_VEL
LIN {X 0,Y 465.355,Z 828.269,A -85,B 0,C 180,E1 14737.393,E2 14737.393} C_VEL
LIN {X 0,Y 461.215,Z 857.701,A -85,B 0,C 180,E1 14736.816,E2 14736.816} C_VEL
LIN {X 0,Y 456.981,Z 880.149,A -85,B 0,C 180,E1 14736.253,E2 14736.253} C_VEL
LIN {X 0,Y 452.314,Z 900.924,A -85,B 0,C 180,E1 14735.608,E2 14735.608} C_VEL
LIN {X 0,Y 446.88,Z 921.805,A -85,B 0,C 180,E1 14734.828,E2 14734.828} C_VEL
LIN {X 0,Y 439.428,Z 946.899,A -85,B 0,C 180,E1 14733.7,E2 14733.7} C_VEL
LIN {X 0,Y 430.983,Z 971.219,A -85,B 0,C 180,E1 14732.354,E2 14732.354} C_VEL
LIN {X 0,Y 423.264,Z 991.389,A -85,B 0,C 180,E1 14731.035,E2 14731.035} C_VEL
LIN {X 0,Y 415.52,Z 1010.052,A -85,B 0,C 180,E1 14729.615,E2 14729.615} C_VEL
LIN {X 0,Y 406.165,Z 1030.964,A -85,B 0,C 180,E1 14727.771,E2 14727.771} C_VEL
LIN {X 0,Y 395.582,Z 1052.648,A -85,B 0,C 180,E1 14725.485,E2 14725.485} C_VEL
LIN {X 0,Y 387.068,Z 1069.132,A -85,B 0,C 180,E1 14723.452,E2 14723.452} C_VEL
LIN {X 0,Y 378.768,Z 1084.535,A -85,B 0,C 180,E1 14721.27,E2 14721.27} C_VEL
LIN {X 0,Y 370.301,Z 1099.759,A -85,B 0,C 180,E1 14718.787,E2 14718.787} C_VEL
LIN {X 0,Y 360.458,Z 1117.155,A -85,B 0,C 180,E1 14715.469,E2 14715.469} C_VEL
LIN {X 0,Y 351.507,Z 1132.488,A -85,B 0,C 180,E1 14711.948,E2 14711.948} C_VEL
LIN {X 0,Y 344.722,Z 1144.272,A -85,B 0,C 180,E1 14708.792,E2 14708.792} C_VEL
LIN {X 0,Y 338.571,Z 1155.302,A -85,B 0,C 180,E1 14705.368,E2 14705.368} C_VEL
LIN {X 0,Y 332.188,Z 1167.414,A -85,B 0,C 180,E1 14700.923,E2 14700.923} C_VEL
LIN {X 0,Y 327.578,Z 1176.885,A -85,B 0,C 180,E1 14696.659,E2 14696.659} C_VEL
LIN {X 0,Y 324.539,Z 1183.995,A -85,B 0,C 180,E1 14692.842,E2 14692.842} C_VEL
LIN {X 0,Y 322.476,Z 1189.682,A -85,B 0,C 180,E1 14689.187,E2 14689.187} C_VEL
LIN {X 0,Y 321.089,Z 1194.556,A -85,B 0,C 180,E1 14685.348,E2 14685.348} C_VEL
LIN {X 0,Y 320.285,Z 1198.503,A -85,B 0,C 180,E1 14681.342,E2 14681.342} C_VEL
LIN {X 0,Y 319.966,Z 1201.642,A -85,B 0,C 180,E1 14676.82,E2 14676.82} C_VEL
LIN {X 0,Y 319.915,Z 1203.137,A -85,B 0,C 180,E1 14672.508,E2 14672.508} C_VEL
LIN {X 0,Y 319.916,Z 1203.398,A -85,B 0,C 180,E1 14668.746,E2 14668.746} C_VEL
LIN {X 0,Y 319.927,Z 1202.653,A -85,B 0,C 180,E1 14664.98,E2 14664.98} C_VEL
LIN {X 0,Y 320.064,Z 1200.905,A -85,B 0,C 180,E1 14661.195,E2 14661.195} C_VEL
LIN {X 0,Y 320.49,Z 1198.154,A -85,B 0,C 180,E1 14657.386,E2 14657.386} C_VEL
LIN {X 0,Y 321.458,Z 1194.388,A -85,B 0,C 180,E1 14653.558,E2 14653.558} C_VEL
LIN {X 0,Y 323.137,Z 1189.486,A -85,B 0,C 180,E1 14649.65,E2 14649.65} C_VEL
LIN {X 0,Y 325.707,Z 1183.478,A -85,B 0,C 180,E1 14645.751,E2 14645.751} C_VEL
LIN {X 0,Y 329.801,Z 1175.344,A -85,B 0,C 180,E1 14641.379,E2 14641.379} C_VEL
LIN {X 0,Y 335.988,Z 1164.343,A -85,B 0,C 180,E1 14636.596,E2 14636.596} C_VEL
LIN {X 0,Y 342.195,Z 1154.161,A -85,B 0,C 180,E1 14632.912,E2 14632.912} C_VEL
LIN {X 0,Y 348.894,Z 1143.608,A -85,B 0,C 180,E1 14629.634,E2 14629.634} C_VEL
LIN {X 0,Y 356.687,Z 1131.546,A -85,B 0,C 180,E1 14626.403,E2 14626.403} C_VEL
LIN {X 0,Y 367.336,Z 1115.179,A -85,B 0,C 180,E1 14622.7,E2 14622.7} C_VEL
LIN {X 0,Y 377.738,Z 1098.742,A -85,B 0,C 180,E1 14619.622,E2 14619.622} C_VEL
LIN {X 0,Y 387.17,Z 1083.491,A -85,B 0,C 180,E1 14617.18,E2 14617.18} C_VEL
LIN {X 0,Y 397.23,Z 1066.628,A -85,B 0,C 180,E1 14614.859,E2 14614.859} C_VEL
LIN {X 0,Y 409.627,Z 1044.584,A -85,B 0,C 180,E1 14612.315,E2 14612.315} C_VEL
LIN {X 0,Y 419.274,Z 1026.127,A -85,B 0,C 180,E1 14610.529,E2 14610.529} C_VEL
LIN {X 0,Y 428.022,Z 1008.265,A -85,B 0,C 180,E1 14609.04,E2 14609.04} C_VEL
LIN {X 0,Y 436.368,Z 989.936,A -85,B 0,C 180,E1 14607.72,E2 14607.72} C_VEL
LIN {X 0,Y 444.618,Z 970.179,A -85,B 0,C 180,E1 14606.489,E2 14606.489} C_VEL
LIN {X 0,Y 454.083,Z 944.998,A -85,B 0,C 180,E1 14605.178,E2 14605.178} C_VEL
LIN {X 0,Y 461.724,Z 921.371,A -85,B 0,C 180,E1 14604.176,E2 14604.176} C_VEL
LIN {X 0,Y 467.561,Z 900.804,A -85,B 0,C 180,E1 14603.452,E2 14603.452} C_VEL
LIN {X 0,Y 472.713,Z 879.766,A -85,B 0,C 180,E1 14602.838,E2 14602.838} C_VEL
LIN {X 0,Y 477.217,Z 857.793,A -85,B 0,C 180,E1 14602.318,E2 14602.318} C_VEL
LIN {X 0,Y 481.672,Z 829.257,A -85,B 0,C 180,E1 14601.783,E2 14601.783} C_VEL
LIN {X 0,Y 486.182,Z 781.402,A -85,B 0,C 180,E1 14601.032,E2 14601.032} C_VEL
LIN {X 0,Y 505.44,Z 566.529,A -85,B 0,C 180,E1 14597.761,E2 14597.761} C_VEL
LIN {X 0,Y 501.406,Z 559.654,A -85,B 0,C 180,E1 14595.44,E2 14595.44} C_VEL
LIN {X 0,Y 498.531,Z 554.952,A -85,B 0,C 180,E1 14593.454,E2 14593.454} C_VEL
LIN {X 0,Y 496.121,Z 550.984,A -85,B 0,C 180,E1 14591.391,E2 14591.391} C_VEL
LIN {X 0,Y 493.64,Z 546.577,A -85,B 0,C 180,E1 14588.386,E2 14588.386} C_VEL
LIN {X 0,Y 491.96,Z 544.755,A -85,B 0,C 180,E1 14583.711,E2 14583.711} C_VEL
LIN {X 0,Y 492.429,Z 545.478,A -85,B 0,C 180,E1 14580.698,E2 14580.698} C_VEL
LIN {X 0,Y 493.85,Z 546.966,A -85,B 0,C 180,E1 14578.086,E2 14578.086} C_VEL
LIN {X 0,Y 496.893,Z 552.221,A -85,B 0,C 180,E1 14574.689,E2 14574.689} C_VEL
LIN {X 0,Y 499.729,Z 556.877,A -85,B 0,C 180,E1 14572.469,E2 14572.469} C_VEL
LIN {X 0,Y 502.897,Z 562.215,A -85,B 0,C 180,E1 14570.443,E2 14570.443} C_VEL
LIN {X 0,Y 505.358,Z 566.495,A -85,B 0,C 180,E1 14569.071,E2 14569.071} C_VEL
LIN {X 0,Y 486.056,Z 781.6,A -85,B 0,C 180,E1 14565.8,E2 14565.8} C_VEL
LIN {X 0,Y 481.723,Z 827.025,A -85,B 0,C 180,E1 14565.085,E2 14565.085} C_VEL
LIN {X 0,Y 477.366,Z 854.555,A -85,B 0,C 180,E1 14564.556,E2 14564.556} C_VEL
LIN {X 0,Y 472.887,Z 876.482,A -85,B 0,C 180,E1 14564.023,E2 14564.023} C_VEL
LIN {X 0,Y 467.711,Z 897.686,A -85,B 0,C 180,E1 14563.386,E2 14563.386} C_VEL
LIN {X 0,Y 461.621,Z 919.127,A -85,B 0,C 180,E1 14562.608,E2 14562.608} C_VEL
LIN {X 0,Y 452.981,Z 945.348,A -85,B 0,C 180,E1 14561.447,E2 14561.447} C_VEL
LIN {X 0,Y 444.57,Z 967.414,A -85,B 0,C 180,E1 14560.258,E2 14560.258} C_VEL
LIN {X 0,Y 436.374,Z 986.926,A -85,B 0,C 180,E1 14559.019,E2 14559.019} C_VEL
LIN {X 0,Y 428.389,Z 1004.423,A -85,B 0,C 180,E1 14557.733,E2 14557.733} C_VEL
LIN {X 0,Y 419.219,Z 1023.037,A -85,B 0,C 180,E1 14556.158,E2 14556.158} C_VEL
LIN {X 0,Y 407.08,Z 1045.85,A -85,B 0,C 180,E1 14553.861,E2 14553.861} C_VEL
LIN {X 0,Y 396.903,Z 1063.55,A -85,B 0,C 180,E1 14551.731,E2 14551.731} C_VEL
LIN {X 0,Y 387.45,Z 1079.24,A -85,B 0,C 180,E1 14549.533,E2 14549.533} C_VEL
LIN {X 0,Y 378.077,Z 1094.218,A -85,B 0,C 180,E1 14547.104,E2 14547.104} C_VEL
LIN {X 0,Y 367.397,Z 1110.918,A -85,B 0,C 180,E1 14543.927,E2 14543.927} C_VEL
LIN {X 0,Y 357.016,Z 1126.555,A -85,B 0,C 180,E1 14540.315,E2 14540.315} C_VEL
LIN {X 0,Y 349.274,Z 1138.291,A -85,B 0,C 180,E1 14537.125,E2 14537.125} C_VEL
LIN {X 0,Y 342.435,Z 1148.842,A -85,B 0,C 180,E1 14533.789,E2 14533.789} C_VEL
LIN {X 0,Y 335.237,Z 1160.553,A -85,B 0,C 180,E1 14529.42,E2 14529.42} C_VEL
LIN {X 0,Y 329.413,Z 1170.527,A -85,B 0,C 180,E1 14524.794,E2 14524.794} C_VEL
LIN {X 0,Y 325.764,Z 1177.617,A -85,B 0,C 180,E1 14520.835,E2 14520.835} C_VEL
LIN {X 0,Y 323.157,Z 1183.511,A -85,B 0,C 180,E1 14516.855,E2 14516.855} C_VEL
LIN {X 0,Y 321.291,Z 1188.884,A -85,B 0,C 180,E1 14512.313,E2 14512.313} C_VEL
LIN {X 0,Y 320.296,Z 1192.982,A -85,B 0,C 180,E1 14507.438,E2 14507.438} C_VEL
LIN {X 0,Y 319.997,Z 1195.113,A -85,B 0,C 180,E1 14503.553,E2 14503.553} C_VEL
LIN {X 0,Y 319.925,Z 1196.198,A -85,B 0,C 180,E1 14499.898,E2 14499.898} C_VEL
LIN {X 0,Y 319.92,Z 1196.37,A -85,B 0,C 180,E1 14496.28,E2 14496.28} C_VEL
LIN {X 0,Y 319.931,Z 1195.643,A -85,B 0,C 180,E1 14492.687,E2 14492.687} C_VEL
LIN {X 0,Y 320.057,Z 1193.913,A -85,B 0,C 180,E1 14488.926,E2 14488.926} C_VEL
LIN {X 0,Y 320.401,Z 1191.361,A -85,B 0,C 180,E1 14485.346,E2 14485.346} C_VEL
LIN {X 0,Y 321.226,Z 1187.704,A -85,B 0,C 180,E1 14481.588,E2 14481.588} C_VEL
LIN {X 0,Y 322.653,Z 1183.034,A -85,B 0,C 180,E1 14477.835,E2 14477.835} C_VEL
LIN {X 0,Y 324.82,Z 1177.325,A -85,B 0,C 180,E1 14474.1,E2 14474.1} C_VEL
LIN {X 0,Y 327.993,Z 1170.194,A -85,B 0,C 180,E1 14470.222,E2 14470.222} C_VEL
LIN {X 0,Y 333.047,Z 1160.222,A -85,B 0,C 180,E1 14465.714,E2 14465.714} C_VEL
LIN {X 0,Y 339.304,Z 1148.67,A -85,B 0,C 180,E1 14461.486,E2 14461.486} C_VEL
LIN {X 0,Y 345.31,Z 1138.149,A -85,B 0,C 180,E1 14458.198,E2 14458.198} C_VEL
LIN {X 0,Y 351.854,Z 1126.95,A -85,B 0,C 180,E1 14455.168,E2 14455.168} C_VEL
LIN {X 0,Y 360.032,Z 1113.104,A -85,B 0,C 180,E1 14451.937,E2 14451.937} C_VEL
LIN {X 0,Y 370.493,Z 1094.996,A -85,B 0,C 180,E1 14448.403,E2 14448.403} C_VEL
LIN {X 0,Y 379.109,Z 1079.654,A -85,B 0,C 180,E1 14445.872,E2 14445.872} C_VEL
LIN {X 0,Y 387.297,Z 1064.574,A -85,B 0,C 180,E1 14443.709,E2 14443.709} C_VEL
LIN {X 0,Y 389.584,Z 1060.327,A -85,B 0,C 180,E1 14443.143,E2 14443.143} C_VEL
LIN {X 0,Y 391.732,Z 1055.133,A -85,B 0,C 180,E1 14442.356,E2 14442.356} C_VEL
LIN {X 0,Y 394.821,Z 1041.552,A -85,B 0,C 180,E1 14440.025,E2 14440.025} C_VEL
LIN {X 0,Y 396.756,Z 1036.692,A -85,B 0,C 180,E1 14439.422,E2 14439.422} C_VEL
LIN {X 0,Y 404.999,Z 1019.721,A -85,B 0,C 180,E1 14437.755,E2 14437.755} C_VEL
LIN {X 0,Y 412.931,Z 1002.284,A -85,B 0,C 180,E1 14436.263,E2 14436.263} C_VEL
LIN {X 0,Y 421.254,Z 982.482,A -85,B 0,C 180,E1 14434.791,E2 14434.791} C_VEL
LIN {X 0,Y 431.163,Z 956.205,A -85,B 0,C 180,E1 14433.16,E2 14433.16} C_VEL
LIN {X 0,Y 438.195,Z 935.087,A -85,B 0,C 180,E1 14432.075,E2 14432.075} C_VEL
LIN {X 0,Y 444.176,Z 914.937,A -85,B 0,C 180,E1 14431.197,E2 14431.197} C_VEL
LIN {X 0,Y 449.524,Z 894.366,A -85,B 0,C 180,E1 14430.437,E2 14430.437} C_VEL
LIN {X 0,Y 454.834,Z 870.487,A -85,B 0,C 180,E1 14429.712,E2 14429.712} C_VEL
LIN {X 0,Y 459.806,Z 841.826,A -85,B 0,C 180,E1 14429.047,E2 14429.047} C_VEL
LIN {X 0,Y 462.686,Z 818.651,A -85,B 0,C 180,E1 14428.626,E2 14428.626} C_VEL
LIN {X 0,Y 479.238,Z 613.765,A -85,B 0,C 180,E1 14425.443,E2 14425.443} C_VEL
LIN {X 0,Y 483.63,Z 560.286,A -85,B 0,C 180,E1 14424.62,E2 14424.62} C_VEL
LIN {X 0,Y 477.8,Z 550.542,A -85,B 0,C 180,E1 14422.226,E2 14422.226} C_VEL
LIN {X 0,Y 472.52,Z 542.058,A -85,B 0,C 180,E1 14419.726,E2 14419.726} C_VEL
LIN {X 0,Y 467.655,Z 534.272,A -85,B 0,C 180,E1 14416.969,E2 14416.969} C_VEL
LIN {X 0,Y 464.523,Z 529.63,A -85,B 0,C 180,E1 14414.842,E2 14414.842} C_VEL
LIN {X 0,Y 461.486,Z 524.98,A -85,B 0,C 180,E1 14412.259,E2 14412.259} C_VEL
LIN {X 0,Y 459.007,Z 520.99,A -85,B 0,C 180,E1 14409.277,E2 14409.277} C_VEL
LIN {X 0,Y 458.566,Z 520.075,A -85,B 0,C 180,E1 14408.527,E2 14408.527} C_VEL
LIN {X 0,Y 457.024,Z 518.874,A -85,B 0,C 180,E1 14403.512,E2 14403.512} C_VEL
LIN {X 0,Y 458.612,Z 520.119,A -85,B 0,C 180,E1 14398.501,E2 14398.501} C_VEL
LIN {X 0,Y 461.295,Z 524.77,A -85,B 0,C 180,E1 14395.026,E2 14395.026} C_VEL
LIN {X 0,Y 462.145,Z 525.929,A -85,B 0,C 180,E1 14394.226,E2 14394.226} C_VEL
LIN {X 0,Y 465.527,Z 531.073,A -85,B 0,C 180,E1 14391.539,E2 14391.539} C_VEL
LIN {X 0,Y 468.788,Z 536.244,A -85,B 0,C 180,E1 14389.43,E2 14389.43} C_VEL
LIN {X 0,Y 472.812,Z 542.456,A -85,B 0,C 180,E1 14387.233,E2 14387.233} C_VEL
LIN {X 0,Y 478.967,Z 552.357,A -85,B 0,C 180,E1 14384.377,E2 14384.377} C_VEL
LIN {X 0,Y 483.703,Z 560.469,A -85,B 0,C 180,E1 14382.453,E2 14382.453} C_VEL
LIN {X 0,Y 466.017,Z 780.198,A -85,B 0,C 180,E1 14379.058,E2 14379.058} C_VEL
LIN {X 0,Y 461.872,Z 828.95,A -85,B 0,C 180,E1 14378.279,E2 14378.279} C_VEL
LIN {X 0,Y 457.691,Z 857.86,A -85,B 0,C 180,E1 14377.713,E2 14377.713} C_VEL
LIN {X 0,Y 453.42,Z 880.086,A -85,B 0,C 180,E1 14377.161,E2 14377.161} C_VEL
LIN {X 0,Y 448.566,Z 901.252,A -85,B 0,C 180,E1 14376.509,E2 14376.509} C_VEL
LIN {X 0,Y 442.699,Z 923.26,A -85,B 0,C 180,E1 14375.689,E2 14375.689} C_VEL
LIN {X 0,Y 434.381,Z 950.095,A -85,B 0,C 180,E1 14374.462,E2 14374.462} C_VEL
LIN {X 0,Y 426.607,Z 971.916,A -85,B 0,C 180,E1 14373.248,E2 14373.248} C_VEL
LIN {X 0,Y 419.041,Z 991.246,A -85,B 0,C 180,E1 14371.987,E2 14371.987} C_VEL
LIN {X 0,Y 411.354,Z 1009.351,A -85,B 0,C 180,E1 14370.62,E2 14370.62} C_VEL
LIN {X 0,Y 402.291,Z 1029.136,A -85,B 0,C 180,E1 14368.895,E2 14368.895} C_VEL
LIN {X 0,Y 390.877,Z 1052.105,A -85,B 0,C 180,E1 14366.501,E2 14366.501} C_VEL
LIN {X 0,Y 381.818,Z 1069.146,A -85,B 0,C 180,E1 14364.399,E2 14364.399} C_VEL
LIN {X 0,Y 373.255,Z 1084.562,A -85,B 0,C 180,E1 14362.207,E2 14362.207} C_VEL
LIN {X 0,Y 364.474,Z 1099.857,A -85,B 0,C 180,E1 14359.697,E2 14359.697} C_VEL
LIN {X 0,Y 354.12,Z 1117.502,A -85,B 0,C 180,E1 14356.287,E2 14356.287} C_VEL
LIN {X 0,Y 345.264,Z 1132.15,A -85,B 0,C 180,E1 14352.886,E2 14352.886} C_VEL
LIN {X 0,Y 338.18,Z 1143.962,A -85,B 0,C 180,E1 14349.689,E2 14349.689} C_VEL
LIN {X 0,Y 331.714,Z 1155.015,A -85,B 0,C 180,E1 14346.213,E2 14346.213} C_VEL
LIN {X 0,Y 325.071,Z 1167.064,A -85,B 0,C 180,E1 14341.733,E2 14341.733} C_VEL
LIN {X 0,Y 320.122,Z 1176.666,A -85,B 0,C 180,E1 14337.331,E2 14337.331} C_VEL
LIN {X 0,Y 316.895,Z 1183.799,A -85,B 0,C 180,E1 14333.425,E2 14333.425} C_VEL
LIN {X 0,Y 314.684,Z 1189.505,A -85,B 0,C 180,E1 14329.682,E2 14329.682} C_VEL
LIN {X 0,Y 313.191,Z 1194.396,A -85,B 0,C 180,E1 14325.745,E2 14325.745} C_VEL
LIN {X 0,Y 312.344,Z 1198.199,A -85,B 0,C 180,E1 14321.822,E2 14321.822} C_VEL
LIN {X 0,Y 312.002,Z 1201.059,A -85,B 0,C 180,E1 14317.735,E2 14317.735} C_VEL
LIN {X 0,Y 311.917,Z 1202.926,A -85,B 0,C 180,E1 14313.308,E2 14313.308} C_VEL
LIN {X 0,Y 311.914,Z 1203.341,A -85,B 0,C 180,E1 14308.898,E2 14308.898} C_VEL
LIN {X 0,Y 311.929,Z 1202.586,A -85,B 0,C 180,E1 14304.851,E2 14304.851} C_VEL
LIN {X 0,Y 312.077,Z 1200.854,A -85,B 0,C 180,E1 14300.968,E2 14300.968} C_VEL
LIN {X 0,Y 312.547,Z 1198.118,A -85,B 0,C 180,E1 14297.06,E2 14297.06} C_VEL
LIN {X 0,Y 313.596,Z 1194.367,A -85,B 0,C 180,E1 14293.134,E2 14293.134} C_VEL
LIN {X 0,Y 315.364,Z 1189.582,A -85,B 0,C 180,E1 14289.201,E2 14289.201} C_VEL
LIN {X 0,Y 318.023,Z 1183.734,A -85,B 0,C 180,E1 14285.282,E2 14285.282} C_VEL
LIN {X 0,Y 321.877,Z 1176.437,A -85,B 0,C 180,E1 14281.218,E2 14281.218} C_VEL
LIN {X 0,Y 328.217,Z 1165.79,A -85,B 0,C 180,E1 14276.328,E2 14276.328} C_VEL
LIN {X 0,Y 335.423,Z 1154.463,A -85,B 0,C 180,E1 14272.116,E2 14272.116} C_VEL
LIN {X 0,Y 342.544,Z 1143.738,A -85,B 0,C 180,E1 14268.725,E2 14268.725} C_VEL
LIN {X 0,Y 350.667,Z 1131.703,A -85,B 0,C 180,E1 14265.459,E2 14265.459} C_VEL
LIN {X 0,Y 361.736,Z 1115.395,A -85,B 0,C 180,E1 14261.73,E2 14261.73} C_VEL
LIN {X 0,Y 372.502,Z 1098.992,A -85,B 0,C 180,E1 14258.639,E2 14258.639} C_VEL
LIN {X 0,Y 381.933,Z 1084.25,A -85,B 0,C 180,E1 14256.263,E2 14256.263} C_VEL
LIN {X 0,Y 391.666,Z 1068.446,A -85,B 0,C 180,E1 14254.066,E2 14254.066} C_VEL
LIN {X 0,Y 403.413,Z 1048.468,A -85,B 0,C 180,E1 14251.699,E2 14251.699} C_VEL
LIN {X 0,Y 415.062,Z 1026.856,A -85,B 0,C 180,E1 14249.585,E2 14249.585} C_VEL
LIN {X 0,Y 424.307,Z 1008.448,A -85,B 0,C 180,E1 14248.056,E2 14248.056} C_VEL
LIN {X 0,Y 432.915,Z 989.995,A -85,B 0,C 180,E1 14246.74,E2 14246.74} C_VEL
LIN {X 0,Y 441.096,Z 970.84,A -85,B 0,C 180,E1 14245.556,E2 14245.556} C_VEL
LIN {X 0,Y 450.374,Z 946.911,A -85,B 0,C 180,E1 14244.31,E2 14244.31} C_VEL
LIN {X 0,Y 458.69,Z 921.819,A -85,B 0,C 180,E1 14243.25,E2 14243.25} C_VEL
LIN {X 0,Y 464.832,Z 900.595,A -85,B 0,C 180,E1 14242.513,E2 14242.513} C_VEL
LIN {X 0,Y 470.024,Z 879.754,A -85,B 0,C 180,E1 14241.914,E2 14241.914} C_VEL
LIN {X 0,Y 474.603,Z 857.793,A -85,B 0,C 180,E1 14241.403,E2 14241.403} C_VEL
LIN {X 0,Y 479.122,Z 829.416,A -85,B 0,C 180,E1 14240.876,E2 14240.876} C_VEL
LIN {X 0,Y 483.711,Z 781.863,A -85,B 0,C 180,E1 14240.134,E2 14240.134} C_VEL
LIN {X 0,Y 502.915,Z 572.266,A -85,B 0,C 180,E1 14236.96,E2 14236.96} C_VEL
LIN {X 0,Y 499.453,Z 566.425,A -85,B 0,C 180,E1 14234.848,E2 14234.848} C_VEL
LIN {X 0,Y 497.178,Z 562.553,A -85,B 0,C 180,E1 14233.195,E2 14233.195} C_VEL
LIN {X 0,Y 495.027,Z 558.871,A -85,B 0,C 180,E1 14231.299,E2 14231.299} C_VEL
LIN {X 0,Y 492.509,Z 554.427,A -85,B 0,C 180,E1 14228.17,E2 14228.17} C_VEL
LIN {X 0,Y 490.981,Z 552.68,A -85,B 0,C 180,E1 14223.62,E2 14223.62} C_VEL
LIN {X 0,Y 491.493,Z 553.475,A -85,B 0,C 180,E1 14220.583,E2 14220.583} C_VEL
LIN {X 0,Y 492.784,Z 554.857,A -85,B 0,C 180,E1 14218.198,E2 14218.198} C_VEL
LIN {X 0,Y 495.706,Z 560.019,A -85,B 0,C 180,E1 14214.85,E2 14214.85} C_VEL
LIN {X 0,Y 498.484,Z 564.7,A -85,B 0,C 180,E1 14212.624,E2 14212.624} C_VEL
LIN {X 0,Y 501.695,Z 570.214,A -85,B 0,C 180,E1 14210.536,E2 14210.536} C_VEL
LIN {X 0,Y 502.837,Z 572.281,A -85,B 0,C 180,E1 14209.869,E2 14209.869} C_VEL
LIN {X 0,Y 483.113,Z 787.401,A -85,B 0,C 180,E1 14206.617,E2 14206.617} C_VEL
LIN {X 0,Y 478.982,Z 828.85,A -85,B 0,C 180,E1 14205.965,E2 14205.965} C_VEL
LIN {X 0,Y 474.596,Z 855.523,A -85,B 0,C 180,E1 14205.452,E2 14205.452} C_VEL
LIN {X 0,Y 470.095,Z 877.074,A -85,B 0,C 180,E1 14204.933,E2 14204.933} C_VEL
LIN {X 0,Y 464.778,Z 898.39,A -85,B 0,C 180,E1 14204.298,E2 14204.298} C_VEL
LIN {X 0,Y 457.919,Z 921.939,A -85,B 0,C 180,E1 14203.445,E2 14203.445} C_VEL
LIN {X 0,Y 449.185,Z 947.386,A -85,B 0,C 180,E1 14202.307,E2 14202.307} C_VEL
LIN {X 0,Y 441.011,Z 968.315,A -85,B 0,C 180,E1 14201.183,E2 14201.183} C_VEL
LIN {X 0,Y 433.027,Z 986.905,A -85,B 0,C 180,E1 14200.011,E2 14200.011} C_VEL
LIN {X 0,Y 424.856,Z 1004.398,A -85,B 0,C 180,E1 14198.74,E2 14198.74} C_VEL
LIN {X 0,Y 415.467,Z 1023.016,A -85,B 0,C 180,E1 14197.179,E2 14197.179} C_VEL
LIN {X 0,Y 403.267,Z 1045.406,A -85,B 0,C 180,E1 14194.948,E2 14194.948} C_VEL
LIN {X 0,Y 392.472,Z 1063.661,A -85,B 0,C 180,E1 14192.761,E2 14192.761} C_VEL
LIN {X 0,Y 382.838,Z 1079.182,A -85,B 0,C 180,E1 14190.592,E2 14190.592} C_VEL
LIN {X 0,Y 373.119,Z 1094.216,A -85,B 0,C 180,E1 14188.154,E2 14188.154} C_VEL
LIN {X 0,Y 361.782,Z 1111.305,A -85,B 0,C 180,E1 14184.89,E2 14184.89} C_VEL
LIN {X 0,Y 351.106,Z 1126.755,A -85,B 0,C 180,E1 14181.286,E2 14181.286} C_VEL
LIN {X 0,Y 343.265,Z 1138.148,A -85,B 0,C 180,E1 14178.16,E2 14178.16} C_VEL
LIN {X 0,Y 336.151,Z 1148.599,A -85,B 0,C 180,E1 14174.824,E2 14174.824} C_VEL
LIN {X 0,Y 329.095,Z 1159.364,A -85,B 0,C 180,E1 14170.784,E2 14170.784} C_VEL
LIN {X 0,Y 322.513,Z 1170.025,A -85,B 0,C 180,E1 14165.869,E2 14165.869} C_VEL
LIN {X 0,Y 318.532,Z 1177.199,A -85,B 0,C 180,E1 14161.826,E2 14161.826} C_VEL
LIN {X 0,Y 315.747,Z 1182.94,A -85,B 0,C 180,E1 14157.929,E2 14157.929} C_VEL
LIN {X 0,Y 313.889,Z 1187.583,A -85,B 0,C 180,E1 14154.062,E2 14154.062} C_VEL
LIN {X 0,Y 312.744,Z 1191.236,A -85,B 0,C 180,E1 14150.199,E2 14150.199} C_VEL
LIN {X 0,Y 312.182,Z 1193.909,A -85,B 0,C 180,E1 14146.37,E2 14146.37} C_VEL
LIN {X 0,Y 311.97,Z 1195.564,A -85,B 0,C 180,E1 14142.776,E2 14142.776} C_VEL
LIN {X 0,Y 311.921,Z 1196.382,A -85,B 0,C 180,E1 14139.223,E2 14139.223} C_VEL
LIN {X 0,Y 311.92,Z 1196.381,A -85,B 0,C 180,E1 14135.703,E2 14135.703} C_VEL
LIN {X 0,Y 311.936,Z 1195.572,A -85,B 0,C 180,E1 14132.204,E2 14132.204} C_VEL
LIN {X 0,Y 312.072,Z 1193.962,A -85,B 0,C 180,E1 14128.715,E2 14128.715} C_VEL
LIN {X 0,Y 312.481,Z 1191.237,A -85,B 0,C 180,E1 14124.86,E2 14124.86} C_VEL
LIN {X 0,Y 313.394,Z 1187.519,A -85,B 0,C 180,E1 14121.006,E2 14121.006} C_VEL
LIN {X 0,Y 314.967,Z 1182.787,A -85,B 0,C 180,E1 14117.161,E2 14117.161} C_VEL
LIN {X 0,Y 317.363,Z 1176.942,A -85,B 0,C 180,E1 14113.294,E2 14113.294} C_VEL
LIN {X 0,Y 321.484,Z 1168.437,A -85,B 0,C 180,E1 14108.661,E2 14108.661} C_VEL
LIN {X 0,Y 327.118,Z 1157.914,A -85,B 0,C 180,E1 14104.082,E2 14104.082} C_VEL
LIN {X 0,Y 332.764,Z 1148.073,A -85,B 0,C 180,E1 14100.477,E2 14100.477} C_VEL
LIN {X 0,Y 339.119,Z 1137.472,A -85,B 0,C 180,E1 14097.146,E2 14097.146} C_VEL
LIN {X 0,Y 346.779,Z 1124.95,A -85,B 0,C 180,E1 14093.767,E2 14093.767} C_VEL
LIN {X 0,Y 357.142,Z 1107.872,A -85,B 0,C 180,E1 14089.916,E2 14089.916} C_VEL
LIN {X 0,Y 365.903,Z 1093.121,A -85,B 0,C 180,E1 14087.124,E2 14087.124} C_VEL
LIN {X 0,Y 374.373,Z 1078.484,A -85,B 0,C 180,E1 14084.731,E2 14084.731} C_VEL
LIN {X 0,Y 383.41,Z 1062.291,A -85,B 0,C 180,E1 14082.438,E2 14082.438} C_VEL
LIN {X 0,Y 394.773,Z 1040.745,A -85,B 0,C 180,E1 14079.852,E2 14079.852} C_VEL
LIN {X 0,Y 396.756,Z 1036.692,A -85,B 0,C 180,E1 14079.422,E2 14079.422} C_VEL
LIN {X 0,Y 398.989,Z 1031.081,A -85,B 0,C 180,E1 14078.717,E2 14078.717} C_VEL
LIN {X 0,Y 402.384,Z 1017.406,A -85,B 0,C 180,E1 14076.66,E2 14076.66} C_VEL
LIN {X 0,Y 404.578,Z 1011.448,A -85,B 0,C 180,E1 14076.029,E2 14076.029} C_VEL
LIN {X 0,Y 414.443,Z 989.015,A -85,B 0,C 180,E1 14074.281,E2 14074.281} C_VEL
LIN {X 0,Y 422.234,Z 969.739,A -85,B 0,C 180,E1 14073.002,E2 14073.002} C_VEL
LIN {X 0,Y 429.285,Z 950.548,A -85,B 0,C 180,E1 14071.901,E2 14071.901} C_VEL
LIN {X 0,Y 436.229,Z 929.606,A -85,B 0,C 180,E1 14070.879,E2 14070.879} C_VEL
LIN {X 0,Y 444.074,Z 902.218,A -85,B 0,C 180,E1 14069.776,E2 14069.776} C_VEL
LIN {X 0,Y 449.72,Z 878.381,A -85,B 0,C 180,E1 14069.013,E2 14069.013} C_VEL
LIN {X 0,Y 453.996,Z 856.741,A -85,B 0,C 180,E1 14068.452,E2 14068.452} C_VEL
LIN {X 0,Y 457.648,Z 833.653,A -85,B 0,C 180,E1 14067.979,E2 14067.979} C_VEL
LIN {X 0,Y 461.159,Z 799.363,A -85,B 0,C 180,E1 14067.404,E2 14067.404} C_VEL
LIN {X 0,Y 479.544,Z 575.857,A -85,B 0,C 180,E1 14063.964,E2 14063.964} C_VEL
LIN {X 0,Y 480.376,Z 565.326,A -85,B 0,C 180,E1 14063.784,E2 14063.784} C_VEL
LIN {X 0,Y 474.184,Z 554.766,A -85,B 0,C 180,E1 14061.071,E2 14061.071} C_VEL
LIN {X 0,Y 468.671,Z 545.915,A -85,B 0,C 180,E1 14058.213,E2 14058.213} C_VEL
LIN {X 0,Y 465.349,Z 540.66,A -85,B 0,C 180,E1 14056.156,E2 14056.156} C_VEL
LIN {X 0,Y 463.221,Z 537.344,A -85,B 0,C 180,E1 14054.629,E2 14054.629} C_VEL
LIN {X 0,Y 460.387,Z 532.865,A -85,B 0,C 180,E1 14052.162,E2 14052.162} C_VEL
LIN {X 0,Y 457.911,Z 528.802,A -85,B 0,C 180,E1 14049.109,E2 14049.109} C_VEL
LIN {X 0,Y 457.518,Z 527.98,A -85,B 0,C 180,E1 14048.42,E2 14048.42} C_VEL
LIN {X 0,Y 456.047,Z 526.815,A -85,B 0,C 180,E1 14043.52,E2 14043.52} C_VEL
LIN {X 0,Y 457.675,Z 528.088,A -85,B 0,C 180,E1 14038.435,E2 14038.435} C_VEL
LIN {X 0,Y 459.81,Z 532.246,A -85,B 0,C 180,E1 14035.51,E2 14035.51} C_VEL
LIN {X 0,Y 460.888,Z 533.602,A -85,B 0,C 180,E1 14034.46,E2 14034.46} C_VEL
LIN {X 0,Y 464.186,Z 538.752,A -85,B 0,C 180,E1 14031.764,E2 14031.764} C_VEL
LIN {X 0,Y 467.48,Z 544.097,A -85,B 0,C 180,E1 14029.587,E2 14029.587} C_VEL
LIN {X 0,Y 471.745,Z 550.755,A -85,B 0,C 180,E1 14027.234,E2 14027.234} C_VEL
LIN {X 0,Y 478.475,Z 561.987,A -85,B 0,C 180,E1 14024.112,E2 14024.112} C_VEL
LIN {X 0,Y 480.483,Z 565.695,A -85,B 0,C 180,E1 14023.269,E2 14023.269} C_VEL
LIN {X 0,Y 462.365,Z 785.681,A -85,B 0,C 180,E1 14019.882,E2 14019.882} C_VEL
LIN {X 0,Y 458.361,Z 830.94,A -85,B 0,C 180,E1 14019.156,E2 14019.156} C_VEL
LIN {X 0,Y 454.148,Z 858.706,A -85,B 0,C 180,E1 14018.609,E2 14018.609} C_VEL
LIN {X 0,Y 449.862,Z 880.516,A -85,B 0,C 180,E1 14018.069,E2 14018.069} C_VEL
LIN {X 0,Y 445.006,Z 901.272,A -85,B 0,C 180,E1 14017.436,E2 14017.436} C_VEL
LIN {X 0,Y 438.992,Z 923.401,A -85,B 0,C 180,E1 14016.618,E2 14016.618} C_VEL
LIN {X 0,Y 430.509,Z 950.183,A -85,B 0,C 180,E1 14015.403,E2 14015.403} C_VEL
LIN {X 0,Y 422.494,Z 972.191,A -85,B 0,C 180,E1 14014.185,E2 14014.185} C_VEL
LIN {X 0,Y 414.75,Z 991.535,A -85,B 0,C 180,E1 14012.927,E2 14012.927} C_VEL
LIN {X 0,Y 406.981,Z 1009.398,A -85,B 0,C 180,E1 14011.585,E2 14011.585} C_VEL
LIN {X 0,Y 397.226,Z 1030.175,A -85,B 0,C 180,E1 14009.772,E2 14009.772} C_VEL
LIN {X 0,Y 385.986,Z 1052.119,A -85,B 0,C 180,E1 14007.476,E2 14007.476} C_VEL
LIN {X 0,Y 376.676,Z 1069.157,A -85,B 0,C 180,E1 14005.373,E2 14005.373} C_VEL
LIN {X 0,Y 367.895,Z 1084.507,A -85,B 0,C 180,E1 14003.183,E2 14003.183} C_VEL
LIN {X 0,Y 358.544,Z 1100.285,A -85,B 0,C 180,E1 14000.575,E2 14000.575} C_VEL
LIN {X 0,Y 347.395,Z 1118.567,A -85,B 0,C 180,E1 13996.974,E2 13996.974} C_VEL
LIN {X 0,Y 338.621,Z 1132.579,A -85,B 0,C 180,E1 13993.66,E2 13993.66} C_VEL
LIN {X 0,Y 331.357,Z 1144.234,A -85,B 0,C 180,E1 13990.448,E2 13990.448} C_VEL
LIN {X 0,Y 324.627,Z 1155.253,A -85,B 0,C 180,E1 13986.913,E2 13986.913} C_VEL
LIN {X 0,Y 317.701,Z 1167.235,A -85,B 0,C 180,E1 13982.345,E2 13982.345} C_VEL
LIN {X 0,Y 312.524,Z 1176.808,A -85,B 0,C 180,E1 13977.846,E2 13977.846} C_VEL
LIN {X 0,Y 309.14,Z 1183.909,A -85,B 0,C 180,E1 13973.847,E2 13973.847} C_VEL
LIN {X 0,Y 306.817,Z 1189.585,A -85,B 0,C 180,E1 13970.009,E2 13970.009} C_VEL
LIN {X 0,Y 305.247,Z 1194.447,A -85,B 0,C 180,E1 13965.971,E2 13965.971} C_VEL
LIN {X 0,Y 304.331,Z 1198.396,A -85,B 0,C 180,E1 13961.736,E2 13961.736} C_VEL
LIN {X 0,Y 303.969,Z 1201.501,A -85,B 0,C 180,E1 13956.99,E2 13956.99} C_VEL
LIN {X 0,Y 303.915,Z 1202.971,A -85,B 0,C 180,E1 13952.451,E2 13952.451} C_VEL
LIN {X 0,Y 303.915,Z 1203.214,A -85,B 0,C 180,E1 13948.492,E2 13948.492} C_VEL
LIN {X 0,Y 303.934,Z 1202.451,A -85,B 0,C 180,E1 13944.526,E2 13944.526} C_VEL
LIN {X 0,Y 304.106,Z 1200.688,A -85,B 0,C 180,E1 13940.538,E2 13940.538} C_VEL
LIN {X 0,Y 304.647,Z 1197.922,A -85,B 0,C 180,E1 13936.525,E2 13936.525} C_VEL
LIN {X 0,Y 305.809,Z 1194.142,A -85,B 0,C 180,E1 13932.494,E2 13932.494} C_VEL
LIN {X 0,Y 307.769,Z 1189.327,A -85,B 0,C 180,E1 13928.463,E2 13928.463} C_VEL
LIN {X 0,Y 310.643,Z 1183.45,A -85,B 0,C 180,E1 13924.45,E2 13924.45} C_VEL
LIN {X 0,Y 315.014,Z 1175.773,A -85,B 0,C 180,E1 13920.111,E2 13920.111} C_VEL
LIN {X 0,Y 322.136,Z 1164.506,A -85,B 0,C 180,E1 13914.956,E2 13914.956} C_VEL
LIN {X 0,Y 329.195,Z 1154.048,A -85,B 0,C 180,E1 13911.039,E2 13911.039} C_VEL
LIN {X 0,Y 336.675,Z 1143.305,A -85,B 0,C 180,E1 13907.612,E2 13907.612} C_VEL
LIN {X 0,Y 345.468,Z 1130.872,A -85,B 0,C 180,E1 13904.229,E2 13904.229} C_VEL
LIN {X 0,Y 357.772,Z 1113.334,A -85,B 0,C 180,E1 13900.275,E2 13900.275} C_VEL
LIN {X 0,Y 367.937,Z 1098.412,A -85,B 0,C 180,E1 13897.486,E2 13897.486} C_VEL
LIN {X 0,Y 377.106,Z 1084.538,A -85,B 0,C 180,E1 13895.251,E2 13895.251} C_VEL
LIN {X 0,Y 387.147,Z 1068.728,A -85,B 0,C 180,E1 13893.05,E2 13893.05} C_VEL
LIN {X 0,Y 398.322,Z 1050.237,A -85,B 0,C 180,E1 13890.854,E2 13890.854} C_VEL
LIN {X 0,Y 411.107,Z 1027.326,A -85,B 0,C 180,E1 13888.599,E2 13888.599} C_VEL
LIN {X 0,Y 420.912,Z 1008.255,A -85,B 0,C 180,E1 13887.027,E2 13887.027} C_VEL
LIN {X 0,Y 429.584,Z 990.067,A -85,B 0,C 180,E1 13885.744,E2 13885.744} C_VEL
LIN {X 0,Y 438.066,Z 970.623,A -85,B 0,C 180,E1 13884.557,E2 13884.557} C_VEL
LIN {X 0,Y 447.769,Z 946.023,A -85,B 0,C 180,E1 13883.3,E2 13883.3} C_VEL
LIN {X 0,Y 456,Z 921.558,A -85,B 0,C 180,E1 13882.286,E2 13882.286} C_VEL
LIN {X 0,Y 462.277,Z 900.218,A -85,B 0,C 180,E1 13881.558,E2 13881.558} C_VEL
LIN {X 0,Y 467.558,Z 879.316,A -85,B 0,C 180,E1 13880.969,E2 13880.969} C_VEL
LIN {X 0,Y 472.308,Z 856.814,A -85,B 0,C 180,E1 13880.457,E2 13880.457} C_VEL
LIN {X 0,Y 477.042,Z 826.506,A -85,B 0,C 180,E1 13879.91,E2 13879.91} C_VEL
LIN {X 0,Y 482.757,Z 767.125,A -85,B 0,C 180,E1 13878.996,E2 13878.996} C_VEL
LIN {X 0,Y 500.48,Z 578.18,A -85,B 0,C 180,E1 13876.156,E2 13876.156} C_VEL
LIN {X 0,Y 496.501,Z 571.067,A -85,B 0,C 180,E1 13873.444,E2 13873.444} C_VEL
LIN {X 0,Y 493.815,Z 566.611,A -85,B 0,C 180,E1 13871.091,E2 13871.091} C_VEL
LIN {X 0,Y 491.46,Z 562.329,A -85,B 0,C 180,E1 13868.07,E2 13868.07} C_VEL
LIN {X 0,Y 490.004,Z 560.623,A -85,B 0,C 180,E1 13863.627,E2 13863.627} C_VEL
LIN {X 0,Y 490.513,Z 561.423,A -85,B 0,C 180,E1 13860.584,E2 13860.584} C_VEL
LIN {X 0,Y 491.72,Z 562.747,A -85,B 0,C 180,E1 13858.31,E2 13858.31} C_VEL
LIN {X 0,Y 494.524,Z 567.817,A -85,B 0,C 180,E1 13855.012,E2 13855.012} C_VEL
LIN {X 0,Y 497.166,Z 572.375,A -85,B 0,C 180,E1 13852.837,E2 13852.837} C_VEL
LIN {X 0,Y 500.414,Z 578.07,A -85,B 0,C 180,E1 13850.678,E2 13850.678} C_VEL
LIN {X 0,Y 480.726,Z 788.274,A -85,B 0,C 180,E1 13847.519,E2 13847.519} C_VEL
LIN {X 0,Y 476.544,Z 829.14,A -85,B 0,C 180,E1 13846.88,E2 13846.88} C_VEL
LIN {X 0,Y 472.12,Z 855.597,A -85,B 0,C 180,E1 13846.378,E2 13846.378} C_VEL
LIN {X 0,Y 467.564,Z 877.062,A -85,B 0,C 180,E1 13845.869,E2 13845.869} C_VEL
LIN {X 0,Y 462.172,Z 898.329,A -85,B 0,C 180,E1 13845.247,E2 13845.247} C_VEL
LIN {X 0,Y 455.191,Z 921.896,A -85,B 0,C 180,E1 13844.406,E2 13844.406} C_VEL
LIN {X 0,Y 446.295,Z 947.362,A -85,B 0,C 180,E1 13843.285,E2 13843.285} C_VEL
LIN {X 0,Y 437.961,Z 968.29,A -85,B 0,C 180,E1 13842.176,E2 13842.176} C_VEL
LIN {X 0,Y 429.554,Z 987.45,A -85,B 0,C 180,E1 13840.981,E2 13840.981} C_VEL
LIN {X 0,Y 420.713,Z 1005.903,A -85,B 0,C 180,E1 13839.645,E2 13839.645} C_VEL
LIN {X 0,Y 409.076,Z 1028.309,A -85,B 0,C 180,E1 13837.737,E2 13837.737} C_VEL
LIN {X 0,Y 397.316,Z 1048.759,A -85,B 0,C 180,E1 13835.624,E2 13835.624} C_VEL
LIN {X 0,Y 387.263,Z 1065.229,A -85,B 0,C 180,E1 13833.624,E2 13833.624} C_VEL
LIN {X 0,Y 377.357,Z 1080.667,A -85,B 0,C 180,E1 13831.444,E2 13831.444} C_VEL
LIN {X 0,Y 366.26,Z 1097.269,A -85,B 0,C 180,E1 13828.7,E2 13828.7} C_VEL
LIN {X 0,Y 354.114,Z 1114.634,A -85,B 0,C 180,E1 13825.223,E2 13825.223} C_VEL
LIN {X 0,Y 344.728,Z 1127.752,A -85,B 0,C 180,E1 13822.084,E2 13822.084} C_VEL
LIN {X 0,Y 336.713,Z 1138.917,A -85,B 0,C 180,E1 13818.959,E2 13818.959} C_VEL
LIN {X 0,Y 328.877,Z 1149.945,A -85,B 0,C 180,E1 13815.35,E2 13815.35} C_VEL
LIN {X 0,Y 320.151,Z 1162.668,A -85,B 0,C 180,E1 13810.276,E2 13810.276} C_VEL
LIN {X 0,Y 314.8,Z 1170.969,A -85,B 0,C 180,E1 13806.211,E2 13806.211} C_VEL
LIN {X 0,Y 310.808,Z 1177.804,A -85,B 0,C 180,E1 13802.211,E2 13802.211} C_VEL
LIN {X 0,Y 307.827,Z 1183.617,A -85,B 0,C 180,E1 13798.098,E2 13798.098} C_VEL
LIN {X 0,Y 305.755,Z 1188.603,A -85,B 0,C 180,E1 13793.699,E2 13793.699} C_VEL
LIN {X 0,Y 304.42,Z 1193.014,A -85,B 0,C 180,E1 13788.379,E2 13788.379} C_VEL
LIN {X 0,Y 304.02,Z 1195.295,A -85,B 0,C 180,E1 13784.015,E2 13784.015} C_VEL
LIN {X 0,Y 303.927,Z 1196.39,A -85,B 0,C 180,E1 13780.041,E2 13780.041} C_VEL
LIN {X 0,Y 303.921,Z 1196.529,A -85,B 0,C 180,E1 13776.233,E2 13776.233} C_VEL
LIN {X 0,Y 303.934,Z 1195.77,A -85,B 0,C 180,E1 13772.451,E2 13772.451} C_VEL
LIN {X 0,Y 304.075,Z 1194.121,A -85,B 0,C 180,E1 13768.681,E2 13768.681} C_VEL
LIN {X 0,Y 304.505,Z 1191.426,A -85,B 0,C 180,E1 13764.725,E2 13764.725} C_VEL
LIN {X 0,Y 305.463,Z 1187.737,A -85,B 0,C 180,E1 13760.771,E2 13760.771} C_VEL
LIN {X 0,Y 307.119,Z 1183.035,A -85,B 0,C 180,E1 13756.827,E2 13756.827} C_VEL
LIN {X 0,Y 309.603,Z 1177.291,A -85,B 0,C 180,E1 13752.91,E2 13752.91} C_VEL
LIN {X 0,Y 313.369,Z 1169.779,A -85,B 0,C 180,E1 13748.67,E2 13748.67} C_VEL
LIN {X 0,Y 319.584,Z 1158.731,A -85,B 0,C 180,E1 13743.624,E2 13743.624} C_VEL
LIN {X 0,Y 325.722,Z 1148.477,A -85,B 0,C 180,E1 13739.773,E2 13739.773} C_VEL
LIN {X 0,Y 332.332,Z 1137.907,A -85,B 0,C 180,E1 13736.387,E2 13736.387} C_VEL
LIN {X 0,Y 340.266,Z 1125.419,A -85,B 0,C 180,E1 13732.959,E2 13732.959} C_VEL
LIN {X 0,Y 351.275,Z 1107.932,A -85,B 0,C 180,E1 13728.966,E2 13728.966} C_VEL
LIN {X 0,Y 360.512,Z 1092.881,A -85,B 0,C 180,E1 13726.104,E2 13726.104} C_VEL
LIN {X 0,Y 369.541,Z 1077.738,A -85,B 0,C 180,E1 13723.628,E2 13723.628} C_VEL
LIN {X 0,Y 380.572,Z 1058.523,A -85,B 0,C 180,E1 13720.946,E2 13720.946} C_VEL
LIN {X 0,Y 391.644,Z 1037.617,A -85,B 0,C 180,E1 13718.532,E2 13718.532} C_VEL
LIN {X 0,Y 400.619,Z 1019.598,A -85,B 0,C 180,E1 13716.761,E2 13716.761} C_VEL
LIN {X 0,Y 404.578,Z 1011.448,A -85,B 0,C 180,E1 13716.029,E2 13716.029} C_VEL
LIN {X 0,Y 406.742,Z 1005.457,A -85,B 0,C 180,E1 13715.414,E2 13715.414} C_VEL
LIN {X 0,Y 410.202,Z 990.783,A -85,B 0,C 180,E1 13713.545,E2 13713.545} C_VEL
LIN {X 0,Y 412.38,Z 984.489,A -85,B 0,C 180,E1 13712.979,E2 13712.979} C_VEL
LIN {X 0,Y 422.026,Z 960.547,A -85,B 0,C 180,E1 13711.471,E2 13711.471} C_VEL
LIN {X 0,Y 430.477,Z 936.331,A -85,B 0,C 180,E1 13710.228,E2 13710.228} C_VEL
LIN {X 0,Y 436.949,Z 915.411,A -85,B 0,C 180,E1 13709.328,E2 13709.328} C_VEL
LIN {X 0,Y 442.489,Z 894.908,A -85,B 0,C 180,E1 13708.583,E2 13708.583} C_VEL
LIN {X 0,Y 447.819,Z 871.877,A -85,B 0,C 180,E1 13707.895,E2 13707.895} C_VEL
LIN {X 0,Y 453.16,Z 842.528,A -85,B 0,C 180,E1 13707.221,E2 13707.221} C_VEL
LIN {X 0,Y 456.193,Z 819.101,A -85,B 0,C 180,E1 13706.8,E2 13706.8} C_VEL
LIN {X 0,Y 473.346,Z 616.648,A -85,B 0,C 180,E1 13703.678,E2 13703.678} C_VEL
LIN {X 0,Y 477.311,Z 570.57,A -85,B 0,C 180,E1 13702.976,E2 13702.976} C_VEL
LIN {X 0,Y 471.602,Z 560.823,A -85,B 0,C 180,E1 13700.348,E2 13700.348} C_VEL
LIN {X 0,Y 466.756,Z 552.863,A -85,B 0,C 180,E1 13697.71,E2 13697.71} C_VEL
LIN {X 0,Y 463.833,Z 548.089,A -85,B 0,C 180,E1 13695.825,E2 13695.825} C_VEL
LIN {X 0,Y 461.926,Z 545.057,A -85,B 0,C 180,E1 13694.414,E2 13694.414} C_VEL
LIN {X 0,Y 459.161,Z 540.623,A -85,B 0,C 180,E1 13691.939,E2 13691.939} C_VEL
LIN {X 0,Y 456.786,Z 536.511,A -85,B 0,C 180,E1 13688.878,E2 13688.878} C_VEL
LIN {X 0,Y 456.396,Z 535.844,A -85,B 0,C 180,E1 13688.187,E2 13688.187} C_VEL
LIN {X 0,Y 455.075,Z 534.748,A -85,B 0,C 180,E1 13683.275,E2 13683.275} C_VEL
LIN {X 0,Y 456.645,Z 536.095,A -85,B 0,C 180,E1 13678.494,E2 13678.494} C_VEL
LIN {X 0,Y 458.826,Z 540.252,A -85,B 0,C 180,E1 13675.5,E2 13675.5} C_VEL
LIN {X 0,Y 459.76,Z 541.535,A -85,B 0,C 180,E1 13674.571,E2 13674.571} C_VEL
LIN {X 0,Y 462.932,Z 546.58,A -85,B 0,C 180,E1 13671.929,E2 13671.929} C_VEL
LIN {X 0,Y 465.98,Z 551.621,A -85,B 0,C 180,E1 13669.866,E2 13669.866} C_VEL
LIN {X 0,Y 470.152,Z 558.303,A -85,B 0,C 180,E1 13667.503,E2 13667.503} C_VEL
LIN {X 0,Y 476.766,Z 569.549,A -85,B 0,C 180,E1 13664.366,E2 13664.366} C_VEL
LIN {X 0,Y 477.372,Z 570.787,A -85,B 0,C 180,E1 13664.097,E2 13664.097} C_VEL
LIN {X 0,Y 458.76,Z 791.781,A -85,B 0,C 180,E1 13660.708,E2 13660.708} C_VEL
LIN {X 0,Y 454.958,Z 832.632,A -85,B 0,C 180,E1 13660.05,E2 13660.05} C_VEL
LIN {X 0,Y 450.778,Z 859.219,A -85,B 0,C 180,E1 13659.526,E2 13659.526} C_VEL
LIN {X 0,Y 446.443,Z 880.82,A -85,B 0,C 180,E1 13658.995,E2 13658.995} C_VEL
LIN {X 0,Y 441.371,Z 902.027,A -85,B 0,C 180,E1 13658.352,E2 13658.352} C_VEL
LIN {X 0,Y 434.646,Z 926.15,A -85,B 0,C 180,E1 13657.459,E2 13657.459} C_VEL
LIN {X 0,Y 426.009,Z 952.322,A -85,B 0,C 180,E1 13656.254,E2 13656.254} C_VEL
LIN {X 0,Y 418.422,Z 972.658,A -85,B 0,C 180,E1 13655.129,E2 13655.129} C_VEL
LIN {X 0,Y 410.416,Z 992.183,A -85,B 0,C 180,E1 13653.862,E2 13653.862} C_VEL
LIN {X 0,Y 402.002,Z 1011.019,A -85,B 0,C 180,E1 13652.443,E2 13652.443} C_VEL
LIN {X 0,Y 390.919,Z 1033.844,A -85,B 0,C 180,E1 13650.414,E2 13650.414} C_VEL
LIN {X 0,Y 380.583,Z 1053.267,A -85,B 0,C 180,E1 13648.343,E2 13648.343} C_VEL
LIN {X 0,Y 371.348,Z 1069.678,A -85,B 0,C 180,E1 13646.303,E2 13646.303} C_VEL
LIN {X 0,Y 362.011,Z 1085.514,A -85,B 0,C 180,E1 13644.023,E2 13644.023} C_VEL
LIN {X 0,Y 351.661,Z 1102.445,A -85,B 0,C 180,E1 13641.173,E2 13641.173} C_VEL
LIN {X 0,Y 340.722,Z 1119.624,A -85,B 0,C 180,E1 13637.689,E2 13637.689} C_VEL
LIN {X 0,Y 332.199,Z 1132.763,A -85,B 0,C 180,E1 13634.53,E2 13634.53} C_VEL
LIN {X 0,Y 324.594,Z 1144.502,A -85,B 0,C 180,E1 13631.238,E2 13631.238} C_VEL
LIN {X 0,Y 317.154,Z 1156.209,A -85,B 0,C 180,E1 13627.393,E2 13627.393} C_VEL
LIN {X 0,Y 309.601,Z 1168.648,A -85,B 0,C 180,E1 13622.418,E2 13622.418} C_VEL
LIN {X 0,Y 304.949,Z 1176.945,A -85,B 0,C 180,E1 13618.387,E2 13618.387} C_VEL
LIN {X 0,Y 301.549,Z 1183.708,A -85,B 0,C 180,E1 13614.486,E2 13614.486} C_VEL
LIN {X 0,Y 299.063,Z 1189.404,A -85,B 0,C 180,E1 13610.551,E2 13610.551} C_VEL
LIN {X 0,Y 297.369,Z 1194.284,A -85,B 0,C 180,E1 13606.406,E2 13606.406} C_VEL
LIN {X 0,Y 296.406,Z 1198.076,A -85,B 0,C 180,E1 13602.27,E2 13602.27} C_VEL
LIN {X 0,Y 296.003,Z 1201.037,A -85,B 0,C 180,E1 13597.765,E2 13597.765} C_VEL
LIN {X 0,Y 295.916,Z 1202.807,A -85,B 0,C 180,E1 13593.099,E2 13593.099} C_VEL
LIN {X 0,Y 295.916,Z 1203.157,A -85,B 0,C 180,E1 13588.645,E2 13588.645} C_VEL
LIN {X 0,Y 295.936,Z 1202.386,A -85,B 0,C 180,E1 13584.377,E2 13584.377} C_VEL
LIN {X 0,Y 296.126,Z 1200.638,A -85,B 0,C 180,E1 13580.281,E2 13580.281} C_VEL
LIN {X 0,Y 296.751,Z 1197.781,A -85,B 0,C 180,E1 13576.027,E2 13576.027} C_VEL
LIN {X 0,Y 297.975,Z 1194.125,A -85,B 0,C 180,E1 13572.019,E2 13572.019} C_VEL
LIN {X 0,Y 300.104,Z 1189.296,A -85,B 0,C 180,E1 13567.857,E2 13567.857} C_VEL
LIN {X 0,Y 303.161,Z 1183.471,A -85,B 0,C 180,E1 13563.772,E2 13563.772} C_VEL
LIN {X 0,Y 307.644,Z 1176.047,A -85,B 0,C 180,E1 13559.462,E2 13559.462} C_VEL
LIN {X 0,Y 315.015,Z 1165.048,A -85,B 0,C 180,E1 13554.267,E2 13554.267} C_VEL
LIN {X 0,Y 322.699,Z 1154.172,A -85,B 0,C 180,E1 13550.106,E2 13550.106} C_VEL
LIN {X 0,Y 330.531,Z 1143.443,A -85,B 0,C 180,E1 13546.633,E2 13546.633} C_VEL
LIN {X 0,Y 339.414,Z 1131.402,A -85,B 0,C 180,E1 13543.313,E2 13543.313} C_VEL
LIN {X 0,Y 351.392,Z 1115.079,A -85,B 0,C 180,E1 13539.547,E2 13539.547} C_VEL
LIN {X 0,Y 362.948,Z 1098.67,A -85,B 0,C 180,E1 13536.447,E2 13536.447} C_VEL
LIN {X 0,Y 372.401,Z 1084.834,A -85,B 0,C 180,E1 13534.214,E2 13534.214} C_VEL
LIN {X 0,Y 382.621,Z 1069.219,A -85,B 0,C 180,E1 13532.039,E2 13532.039} C_VEL
LIN {X 0,Y 393.51,Z 1051.707,A -85,B 0,C 180,E1 13529.953,E2 13529.953} C_VEL
LIN {X 0,Y 406.708,Z 1028.865,A -85,B 0,C 180,E1 13527.688,E2 13527.688} C_VEL
LIN {X 0,Y 417.295,Z 1008.784,A -85,B 0,C 180,E1 13526.037,E2 13526.037} C_VEL
LIN {X 0,Y 426.517,Z 989.872,A -85,B 0,C 180,E1 13524.716,E2 13524.716} C_VEL
LIN {X 0,Y 435.174,Z 970.418,A -85,B 0,C 180,E1 13523.546,E2 13523.546} C_VEL
LIN {X 0,Y 444.972,Z 946.039,A -85,B 0,C 180,E1 13522.319,E2 13522.319} C_VEL
LIN {X 0,Y 453.443,Z 921.301,A -85,B 0,C 180,E1 13521.311,E2 13521.311} C_VEL
LIN {X 0,Y 459.589,Z 900.809,A -85,B 0,C 180,E1 13520.623,E2 13520.623} C_VEL
LIN {X 0,Y 465.019,Z 879.758,A -85,B 0,C 180,E1 13520.036,E2 13520.036} C_VEL
LIN {X 0,Y 469.747,Z 857.838,A -85,B 0,C 180,E1 13519.543,E2 13519.543} C_VEL
LIN {X 0,Y 474.403,Z 829.723,A -85,B 0,C 180,E1 13519.034,E2 13519.034} C_VEL
LIN {X 0,Y 479.101,Z 783.263,A -85,B 0,C 180,E1 13518.318,E2 13518.318} C_VEL
LIN {X 0,Y 498.137,Z 584.137,A -85,B 0,C 180,E1 13515.342,E2 13515.342} C_VEL
LIN {X 0,Y 494.714,Z 578.07,A -85,B 0,C 180,E1 13512.846,E2 13512.846} C_VEL
LIN {X 0,Y 492.609,Z 574.35,A -85,B 0,C 180,E1 13510.881,E2 13510.881} C_VEL
LIN {X 0,Y 490.414,Z 570.231,A -85,B 0,C 180,E1 13507.969,E2 13507.969} C_VEL
LIN {X 0,Y 489.027,Z 568.566,A -85,B 0,C 180,E1 13503.634,E2 13503.634} C_VEL
LIN {X 0,Y 489.534,Z 569.372,A -85,B 0,C 180,E1 13500.585,E2 13500.585} C_VEL
LIN {X 0,Y 490.625,Z 570.534,A -85,B 0,C 180,E1 13498.482,E2 13498.482} C_VEL
LIN {X 0,Y 493.346,Z 575.614,A -85,B 0,C 180,E1 13495.175,E2 13495.175} C_VEL
LIN {X 0,Y 495.93,Z 580.195,A -85,B 0,C 180,E1 13492.994,E2 13492.994} C_VEL
LIN {X 0,Y 498.074,Z 584.144,A -85,B 0,C 180,E1 13491.486,E2 13491.486} C_VEL
LIN {X 0,Y 477.265,Z 802,A -85,B 0,C 180,E1 13488.236,E2 13488.236} C_VEL
LIN {X 0,Y 473.459,Z 834.324,A -85,B 0,C 180,E1 13487.717,E2 13487.717} C_VEL
LIN {X 0,Y 469.494,Z 857.082,A -85,B 0,C 180,E1 13487.283,E2 13487.283} C_VEL
LIN {X 0,Y 464.873,Z 878.287,A -85,B 0,C 180,E1 13486.783,E2 13486.783} C_VEL
LIN {X 0,Y 459.13,Z 900.346,A -85,B 0,C 180,E1 13486.139,E2 13486.139} C_VEL
LIN {X 0,Y 450.935,Z 926.867,A -85,B 0,C 180,E1 13485.181,E2 13485.181} C_VEL
LIN {X 0,Y 442.721,Z 949.418,A -85,B 0,C 180,E1 13484.174,E2 13484.174} C_VEL
LIN {X 0,Y 434.646,Z 969.208,A -85,B 0,C 180,E1 13483.129,E2 13483.129} C_VEL
LIN {X 0,Y 426.151,Z 988.122,A -85,B 0,C 180,E1 13481.958,E2 13481.958} C_VEL
LIN {X 0,Y 417.056,Z 1006.648,A -85,B 0,C 180,E1 13480.627,E2 13480.627} C_VEL
LIN {X 0,Y 405.091,Z 1029.062,A -85,B 0,C 180,E1 13478.725,E2 13478.725} C_VEL
LIN {X 0,Y 393.161,Z 1049.274,A -85,B 0,C 180,E1 13476.645,E2 13476.645} C_VEL
LIN {X 0,Y 382.817,Z 1065.754,A -85,B 0,C 180,E1 13474.648,E2 13474.648} C_VEL
LIN {X 0,Y 372.319,Z 1081.629,A -85,B 0,C 180,E1 13472.401,E2 13472.401} C_VEL
LIN {X 0,Y 360.021,Z 1099.43,A -85,B 0,C 180,E1 13469.422,E2 13469.422} C_VEL
LIN {X 0,Y 348.154,Z 1115.665,A -85,B 0,C 180,E1 13466.096,E2 13466.096} C_VEL
LIN {X 0,Y 338.904,Z 1128.096,A -85,B 0,C 180,E1 13463.084,E2 13463.084} C_VEL
LIN {X 0,Y 330.131,Z 1139.825,A -85,B 0,C 180,E1 13459.749,E2 13459.749} C_VEL
LIN {X 0,Y 320.525,Z 1152.846,A -85,B 0,C 180,E1 13455.335,E2 13455.335} C_VEL
LIN {X 0,Y 312.586,Z 1163.795,A -85,B 0,C 180,E1 13450.702,E2 13450.702} C_VEL
LIN {X 0,Y 307.334,Z 1171.553,A -85,B 0,C 180,E1 13446.77,E2 13446.77} C_VEL
LIN {X 0,Y 303.206,Z 1178.223,A -85,B 0,C 180,E1 13442.739,E2 13442.739} C_VEL
LIN {X 0,Y 299.9,Z 1184.318,A -85,B 0,C 180,E1 13438.257,E2 13438.257} C_VEL
LIN {X 0,Y 297.423,Z 1190.083,A -85,B 0,C 180,E1 13432.743,E2 13432.743} C_VEL
LIN {X 0,Y 296.38,Z 1193.487,A -85,B 0,C 180,E1 13428.081,E2 13428.081} C_VEL
LIN {X 0,Y 296.024,Z 1195.452,A -85,B 0,C 180,E1 13424.075,E2 13424.075} C_VEL
LIN {X 0,Y 295.928,Z 1196.486,A -85,B 0,C 180,E1 13420.119,E2 13420.119} C_VEL
LIN {X 0,Y 295.922,Z 1196.608,A -85,B 0,C 180,E1 13416.207,E2 13416.207} C_VEL
LIN {X 0,Y 295.936,Z 1195.833,A -85,B 0,C 180,E1 13412.324,E2 13412.324} C_VEL
LIN {X 0,Y 296.091,Z 1194.168,A -85,B 0,C 180,E1 13408.452,E2 13408.452} C_VEL
LIN {X 0,Y 296.566,Z 1191.456,A -85,B 0,C 180,E1 13404.389,E2 13404.389} C_VEL
LIN {X 0,Y 297.538,Z 1187.953,A -85,B 0,C 180,E1 13400.523,E2 13400.523} C_VEL
LIN {X 0,Y 299.29,Z 1183.258,A -85,B 0,C 180,E1 13396.458,E2 13396.458} C_VEL
LIN {X 0,Y 301.89,Z 1177.567,A -85,B 0,C 180,E1 13392.459,E2 13392.459} C_VEL
LIN {X 0,Y 305.661,Z 1170.391,A -85,B 0,C 180,E1 13388.285,E2 13388.285} C_VEL
LIN {X 0,Y 311.814,Z 1159.995,A -85,B 0,C 180,E1 13383.326,E2 13383.326} C_VEL
LIN {X 0,Y 318.734,Z 1148.876,A -85,B 0,C 180,E1 13379.039,E2 13379.039} C_VEL
LIN {X 0,Y 325.606,Z 1138.339,A -85,B 0,C 180,E1 13375.596,E2 13375.596} C_VEL
LIN {X 0,Y 333.408,Z 1126.506,A -85,B 0,C 180,E1 13372.282,E2 13372.282} C_VEL
LIN {X 0,Y 343.517,Z 1111.201,A -85,B 0,C 180,E1 13368.646,E2 13368.646} C_VEL
LIN {X 0,Y 354.221,Z 1094.287,A -85,B 0,C 180,E1 13365.344,E2 13365.344} C_VEL
LIN {X 0,Y 363.191,Z 1079.737,A -85,B 0,C 180,E1 13362.921,E2 13362.921} C_VEL
LIN {X 0,Y 372.447,Z 1064.128,A -85,B 0,C 180,E1 13360.678,E2 13360.678} C_VEL
LIN {X 0,Y 382.805,Z 1045.761,A -85,B 0,C 180,E1 13358.411,E2 13358.411} C_VEL
LIN {X 0,Y 394.619,Z 1023.038,A -85,B 0,C 180,E1 13356.074,E2 13356.074} C_VEL
LIN {X 0,Y 403.379,Z 1004.822,A -85,B 0,C 180,E1 13354.496,E2 13354.496} C_VEL
LIN {X 0,Y 411.335,Z 986.916,A -85,B 0,C 180,E1 13353.147,E2 13353.147} C_VEL
LIN {X 0,Y 412.38,Z 984.489,A -85,B 0,C 180,E1 13352.979,E2 13352.979} C_VEL
LIN {X 0,Y 414.65,Z 978.183,A -85,B 0,C 180,E1 13352.431,E2 13352.431} C_VEL
LIN {X 0,Y 418,Z 962.674,A -85,B 0,C 180,E1 13350.729,E2 13350.729} C_VEL
LIN {X 0,Y 419.986,Z 956.086,A -85,B 0,C 180,E1 13350.241,E2 13350.241} C_VEL
LIN {X 0,Y 427.282,Z 935.438,A -85,B 0,C 180,E1 13349.211,E2 13349.211} C_VEL
LIN {X 0,Y 433.547,Z 915.515,A -85,B 0,C 180,E1 13348.366,E2 13348.366} C_VEL
LIN {X 0,Y 439.252,Z 894.769,A -85,B 0,C 180,E1 13347.621,E2 13347.621} C_VEL
LIN {X 0,Y 444.842,Z 870.976,A -85,B 0,C 180,E1 13346.923,E2 13346.923} C_VEL
LIN {X 0,Y 450.107,Z 842.231,A -85,B 0,C 180,E1 13346.276,E2 13346.276} C_VEL
LIN {X 0,Y 453.157,Z 818.983,A -85,B 0,C 180,E1 13345.863,E2 13345.863} C_VEL
LIN {X 0,Y 470.819,Z 615.246,A -85,B 0,C 180,E1 13342.736,E2 13342.736} C_VEL
LIN {X 0,Y 474.219,Z 575.709,A -85,B 0,C 180,E1 13342.109,E2 13342.109} C_VEL
LIN {X 0,Y 468.432,Z 565.605,A -85,B 0,C 180,E1 13339.256,E2 13339.256} C_VEL
LIN {X 0,Y 463.306,Z 556.998,A -85,B 0,C 180,E1 13336.165,E2 13336.165} C_VEL
LIN {X 0,Y 460.636,Z 552.769,A -85,B 0,C 180,E1 13334.199,E2 13334.199} C_VEL
LIN {X 0,Y 458.067,Z 548.509,A -85,B 0,C 180,E1 13331.841,E2 13331.841} C_VEL
LIN {X 0,Y 455.699,Z 544.323,A -85,B 0,C 180,E1 13328.708,E2 13328.708} C_VEL
LIN {X 0,Y 455.141,Z 543.638,A -85,B 0,C 180,E1 13327.701,E2 13327.701} C_VEL
LIN {X 0,Y 454.103,Z 542.685,A -85,B 0,C 180,E1 13323.156,E2 13323.156} C_VEL
LIN {X 0,Y 455.616,Z 544.099,A -85,B 0,C 180,E1 13318.554,E2 13318.554} C_VEL
LIN {X 0,Y 457.842,Z 548.252,A -85,B 0,C 180,E1 13315.491,E2 13315.491} C_VEL
LIN {X 0,Y 458.756,Z 549.716,A -85,B 0,C 180,E1 13314.56,E2 13314.56} C_VEL
LIN {X 0,Y 461.603,Z 554.257,A -85,B 0,C 180,E1 13312.157,E2 13312.157} C_VEL
LIN {X 0,Y 464.776,Z 559.629,A -85,B 0,C 180,E1 13309.964,E2 13309.964} C_VEL
LIN {X 0,Y 468.624,Z 565.954,A -85,B 0,C 180,E1 13307.743,E2 13307.743} C_VEL
LIN {X 0,Y 474.349,Z 575.969,A -85,B 0,C 180,E1 13304.935,E2 13304.935} C_VEL
LIN {X 0,Y 455.204,Z 798.367,A -85,B 0,C 180,E1 13301.54,E2 13301.54} C_VEL
LIN {X 0,Y 451.528,Z 834.941,A -85,B 0,C 180,E1 13300.943,E2 13300.943} C_VEL
LIN {X 0,Y 447.519,Z 859.757,A -85,B 0,C 180,E1 13300.455,E2 13300.455} C_VEL
LIN {X 0,Y 443.163,Z 881.034,A -85,B 0,C 180,E1 13299.937,E2 13299.937} C_VEL
LIN {X 0,Y 437.924,Z 902.5,A -85,B 0,C 180,E1 13299.292,E2 13299.292} C_VEL
LIN {X 0,Y 430.45,Z 928.649,A -85,B 0,C 180,E1 13298.325,E2 13298.325} C_VEL
LIN {X 0,Y 421.983,Z 953.418,A -85,B 0,C 180,E1 13297.176,E2 13297.176} C_VEL
LIN {X 0,Y 414.462,Z 973.121,A -85,B 0,C 180,E1 13296.09,E2 13296.09} C_VEL
LIN {X 0,Y 406.456,Z 992.23,A -85,B 0,C 180,E1 13294.858,E2 13294.858} C_VEL
LIN {X 0,Y 397.616,Z 1011.56,A -85,B 0,C 180,E1 13293.409,E2 13293.409} C_VEL
LIN {X 0,Y 385.493,Z 1035.724,A -85,B 0,C 180,E1 13291.243,E2 13291.243} C_VEL
LIN {X 0,Y 375.589,Z 1053.842,A -85,B 0,C 180,E1 13289.301,E2 13289.301} C_VEL
LIN {X 0,Y 366.121,Z 1070.2,A -85,B 0,C 180,E1 13287.26,E2 13287.26} C_VEL
LIN {X 0,Y 356.532,Z 1085.982,A -85,B 0,C 180,E1 13284.973,E2 13284.973} C_VEL
LIN {X 0,Y 344.811,Z 1104.542,A -85,B 0,C 180,E1 13281.797,E2 13281.797} C_VEL
LIN {X 0,Y 334.103,Z 1120.68,A -85,B 0,C 180,E1 13278.431,E2 13278.431} C_VEL
LIN {X 0,Y 325.772,Z 1133.061,A -85,B 0,C 180,E1 13275.402,E2 13275.402} C_VEL
LIN {X 0,Y 317.893,Z 1144.768,A -85,B 0,C 180,E1 13272.062,E2 13272.062} C_VEL
LIN {X 0,Y 309.618,Z 1157.3,A -85,B 0,C 180,E1 13267.848,E2 13267.848} C_VEL
LIN {X 0,Y 302.274,Z 1168.815,A -85,B 0,C 180,E1 13263.078,E2 13263.078} C_VEL
LIN {X 0,Y 297.403,Z 1177.082,A -85,B 0,C 180,E1 13258.955,E2 13258.955} C_VEL
LIN {X 0,Y 293.834,Z 1183.814,A -85,B 0,C 180,E1 13254.957,E2 13254.957} C_VEL
LIN {X 0,Y 291.116,Z 1189.74,A -85,B 0,C 180,E1 13250.717,E2 13250.717} C_VEL
LIN {X 0,Y 289.311,Z 1194.754,A -85,B 0,C 180,E1 13246.256,E2 13246.256} C_VEL
LIN {X 0,Y 288.239,Z 1199.189,A -85,B 0,C 180,E1 13240.971,E2 13240.971} C_VEL
LIN {X 0,Y 287.95,Z 1201.698,A -85,B 0,C 180,E1 13236.179,E2 13236.179} C_VEL
LIN {X 0,Y 287.914,Z 1202.826,A -85,B 0,C 180,E1 13232.189,E2 13232.189} C_VEL
LIN {X 0,Y 287.914,Z 1203.031,A -85,B 0,C 180,E1 13228.209,E2 13228.209} C_VEL
LIN {X 0,Y 287.945,Z 1202.252,A -85,B 0,C 180,E1 13224.021,E2 13224.021} C_VEL
LIN {X 0,Y 288.17,Z 1200.474,A -85,B 0,C 180,E1 13219.808,E2 13219.808} C_VEL
LIN {X 0,Y 288.856,Z 1197.694,A -85,B 0,C 180,E1 13215.568,E2 13215.568} C_VEL
LIN {X 0,Y 290.248,Z 1193.903,A -85,B 0,C 180,E1 13211.315,E2 13211.315} C_VEL
LIN {X 0,Y 292.565,Z 1189.078,A -85,B 0,C 180,E1 13207.07,E2 13207.07} C_VEL
LIN {X 0,Y 296.103,Z 1182.89,A -85,B 0,C 180,E1 13202.662,E2 13202.662} C_VEL
LIN {X 0,Y 302.16,Z 1173.723,A -85,B 0,C 180,E1 13197.359,E2 13197.359} C_VEL
LIN {X 0,Y 309.547,Z 1163.316,A -85,B 0,C 180,E1 13192.609,E2 13192.609} C_VEL
LIN {X 0,Y 316.685,Z 1153.777,A -85,B 0,C 180,E1 13188.951,E2 13188.951} C_VEL
LIN {X 0,Y 324.935,Z 1143.015,A -85,B 0,C 180,E1 13185.446,E2 13185.446} C_VEL
LIN {X 0,Y 334.728,Z 1130.316,A -85,B 0,C 180,E1 13181.946,E2 13181.946} C_VEL
LIN {X 0,Y 347.784,Z 1113.027,A -85,B 0,C 180,E1 13178.026,E2 13178.026} C_VEL
LIN {X 0,Y 358.67,Z 1098.101,A -85,B 0,C 180,E1 13175.236,E2 13175.236} C_VEL
LIN {X 0,Y 368.448,Z 1084.218,A -85,B 0,C 180,E1 13173.015,E2 13173.015} C_VEL
LIN {X 0,Y 378.727,Z 1068.949,A -85,B 0,C 180,E1 13170.906,E2 13170.906} C_VEL
LIN {X 0,Y 389.488,Z 1052.088,A -85,B 0,C 180,E1 13168.91,E2 13168.91} C_VEL
LIN {X 0,Y 402.861,Z 1029.589,A -85,B 0,C 180,E1 13166.686,E2 13166.686} C_VEL
LIN {X 0,Y 413.988,Z 1008.973,A -85,B 0,C 180,E1 13165.003,E2 13165.003} C_VEL
LIN {X 0,Y 423.21,Z 990.476,A -85,B 0,C 180,E1 13163.725,E2 13163.725} C_VEL
LIN {X 0,Y 431.705,Z 971.84,A -85,B 0,C 180,E1 13162.612,E2 13162.612} C_VEL
LIN {X 0,Y 440.254,Z 951.188,A -85,B 0,C 180,E1 13161.564,E2 13161.564} C_VEL
LIN {X 0,Y 449.819,Z 924.833,A -85,B 0,C 180,E1 13160.462,E2 13160.462} C_VEL
LIN {X 0,Y 456.813,Z 902.165,A -85,B 0,C 180,E1 13159.699,E2 13159.699} C_VEL
LIN {X 0,Y 462.426,Z 880.943,A -85,B 0,C 180,E1 13159.112,E2 13159.112} C_VEL
LIN {X 0,Y 467.146,Z 859.659,A -85,B 0,C 180,E1 13158.635,E2 13158.635} C_VEL
LIN {X 0,Y 471.406,Z 835.43,A -85,B 0,C 180,E1 13158.193,E2 13158.193} C_VEL
LIN {X 0,Y 475.522,Z 799.323,A -85,B 0,C 180,E1 13157.625,E2 13157.625} C_VEL
LIN {X 0,Y 495.897,Z 590.164,A -85,B 0,C 180,E1 13154.524,E2 13154.524} C_VEL
LIN {X 0,Y 493.32,Z 585.561,A -85,B 0,C 180,E1 13152.526,E2 13152.526} C_VEL
LIN {X 0,Y 491.382,Z 582.051,A -85,B 0,C 180,E1 13150.642,E2 13150.642} C_VEL
LIN {X 0,Y 489.369,Z 578.132,A -85,B 0,C 180,E1 13147.868,E2 13147.868} C_VEL
LIN {X 0,Y 488.048,Z 576.489,A -85,B 0,C 180,E1 13143.524,E2 13143.524} C_VEL
LIN {X 0,Y 488.643,Z 577.442,A -85,B 0,C 180,E1 13140.352,E2 13140.352} C_VEL
LIN {X 0,Y 489.566,Z 578.421,A -85,B 0,C 180,E1 13138.596,E2 13138.596} C_VEL
LIN {X 0,Y 492.17,Z 583.411,A -85,B 0,C 180,E1 13135.339,E2 13135.339} C_VEL
LIN {X 0,Y 494.697,Z 588.015,A -85,B 0,C 180,E1 13133.151,E2 13133.151} C_VEL
LIN {X 0,Y 495.833,Z 590.217,A -85,B 0,C 180,E1 13132.303,E2 13132.303} C_VEL
LIN {X 0,Y 474.297,Z 810.884,A -85,B 0,C 180,E1 13129.035,E2 13129.035} C_VEL
LIN {X 0,Y 470.925,Z 836.707,A -85,B 0,C 180,E1 13128.614,E2 13128.614} C_VEL
LIN {X 0,Y 466.991,Z 858.548,A -85,B 0,C 180,E1 13128.199,E2 13128.199} C_VEL
LIN {X 0,Y 462.151,Z 880.142,A -85,B 0,C 180,E1 13127.691,E2 13127.691} C_VEL
LIN {X 0,Y 455.142,Z 906.177,A -85,B 0,C 180,E1 13126.922,E2 13126.922} C_VEL
LIN {X 0,Y 446.755,Z 931.521,A -85,B 0,C 180,E1 13125.975,E2 13125.975} C_VEL
LIN {X 0,Y 439.297,Z 951.375,A -85,B 0,C 180,E1 13125.081,E2 13125.081} C_VEL
LIN {X 0,Y 431.453,Z 970.126,A -85,B 0,C 180,E1 13124.097,E2 13124.097} C_VEL
LIN {X 0,Y 422.597,Z 989.382,A -85,B 0,C 180,E1 13122.912,E2 13122.912} C_VEL
LIN {X 0,Y 411.98,Z 1010.44,A -85,B 0,C 180,E1 13121.392,E2 13121.392} C_VEL
LIN {X 0,Y 399.397,Z 1032.877,A -85,B 0,C 180,E1 13119.435,E2 13119.435} C_VEL
LIN {X 0,Y 388.808,Z 1050.315,A -85,B 0,C 180,E1 13117.628,E2 13117.628} C_VEL
LIN {X 0,Y 378.249,Z 1066.662,A -85,B 0,C 180,E1 13115.645,E2 13115.645} C_VEL
LIN {X 0,Y 366.915,Z 1083.28,A -85,B 0,C 180,E1 13113.279,E2 13113.279} C_VEL
LIN {X 0,Y 353.219,Z 1102.226,A -85,B 0,C 180,E1 13110.019,E2 13110.019} C_VEL
LIN {X 0,Y 342.226,Z 1116.764,A -85,B 0,C 180,E1 13106.983,E2 13106.983} C_VEL
LIN {X 0,Y 332.685,Z 1129.1,A -85,B 0,C 180,E1 13103.945,E2 13103.945} C_VEL
LIN {X 0,Y 322.724,Z 1141.91,A -85,B 0,C 180,E1 13100.206,E2 13100.206} C_VEL
LIN {X 0,Y 312.512,Z 1155,A -85,B 0,C 180,E1 13095.517,E2 13095.517} C_VEL
LIN {X 0,Y 305.419,Z 1164.405,A -85,B 0,C 180,E1 13091.398,E2 13091.398} C_VEL
LIN {X 0,Y 299.9,Z 1172.141,A -85,B 0,C 180,E1 13087.357,E2 13087.357} C_VEL
LIN {X 0,Y 295.206,Z 1179.355,A -85,B 0,C 180,E1 13082.814,E2 13082.814} C_VEL
LIN {X 0,Y 291.163,Z 1186.62,A -85,B 0,C 180,E1 13076.955,E2 13076.955} C_VEL
LIN {X 0,Y 289.297,Z 1190.877,A -85,B 0,C 180,E1 13072.345,E2 13072.345} C_VEL
LIN {X 0,Y 288.395,Z 1193.732,A -85,B 0,C 180,E1 13068.181,E2 13068.181} C_VEL
LIN {X 0,Y 288.035,Z 1195.566,A -85,B 0,C 180,E1 13064.268,E2 13064.268} C_VEL
LIN {X 0,Y 287.932,Z 1196.561,A -85,B 0,C 180,E1 13060.403,E2 13060.403} C_VEL
LIN {X 0,Y 287.919,Z 1196.71,A -85,B 0,C 180,E1 13056.38,E2 13056.38} C_VEL
LIN {X 0,Y 287.935,Z 1195.962,A -85,B 0,C 180,E1 13052.388,E2 13052.388} C_VEL
LIN {X 0,Y 288.095,Z 1194.325,A -85,B 0,C 180,E1 13048.409,E2 13048.409} C_VEL
LIN {X 0,Y 288.594,Z 1191.642,A -85,B 0,C 180,E1 13044.234,E2 13044.234} C_VEL
LIN {X 0,Y 289.689,Z 1187.966,A -85,B 0,C 180,E1 13040.063,E2 13040.063} C_VEL
LIN {X 0,Y 291.562,Z 1183.276,A -85,B 0,C 180,E1 13035.908,E2 13035.908} C_VEL
LIN {X 0,Y 294.343,Z 1177.544,A -85,B 0,C 180,E1 13031.789,E2 13031.789} C_VEL
LIN {X 0,Y 298.333,Z 1170.388,A -85,B 0,C 180,E1 13027.538,E2 13027.538} C_VEL
LIN {X 0,Y 304.851,Z 1159.912,A -85,B 0,C 180,E1 13022.454,E2 13022.454} C_VEL
LIN {X 0,Y 312.15,Z 1148.755,A -85,B 0,C 180,E1 13018.088,E2 13018.088} C_VEL
LIN {X 0,Y 319.325,Z 1138.21,A -85,B 0,C 180,E1 13014.601,E2 13014.601} C_VEL
LIN {X 0,Y 327.451,Z 1126.349,A -85,B 0,C 180,E1 13011.248,E2 13011.248} C_VEL
LIN {X 0,Y 338.428,Z 1110.25,A -85,B 0,C 180,E1 13007.425,E2 13007.425} C_VEL
LIN {X 0,Y 349.042,Z 1094.04,A -85,B 0,C 180,E1 13004.263,E2 13004.263} C_VEL
LIN {X 0,Y 358.315,Z 1079.433,A -85,B 0,C 180,E1 13001.832,E2 13001.832} C_VEL
LIN {X 0,Y 368.133,Z 1063.315,A -85,B 0,C 180,E1 12999.525,E2 12999.525} C_VEL
LIN {X 0,Y 380.049,Z 1042.619,A -85,B 0,C 180,E1 12997.016,E2 12997.016} C_VEL
LIN {X 0,Y 390.814,Z 1022.163,A -85,B 0,C 180,E1 12994.967,E2 12994.967} C_VEL
LIN {X 0,Y 399.59,Z 1004.294,A -85,B 0,C 180,E1 12993.438,E2 12993.438} C_VEL
LIN {X 0,Y 407.974,Z 985.781,A -85,B 0,C 180,E1 12992.064,E2 12992.064} C_VEL
LIN {X 0,Y 416.514,Z 965.153,A -85,B 0,C 180,E1 12990.752,E2 12990.752} C_VEL
LIN {X 0,Y 419.986,Z 956.086,A -85,B 0,C 180,E1 12990.241,E2 12990.241} C_VEL
LIN {X 0,Y 422.027,Z 949.415,A -85,B 0,C 180,E1 12989.773,E2 12989.773} C_VEL
LIN {X 0,Y 425.387,Z 932.138,A -85,B 0,C 180,E1 12988.168,E2 12988.168} C_VEL
LIN {X 0,Y 427.024,Z 926.273,A -85,B 0,C 180,E1 12987.813,E2 12987.813} C_VEL
LIN {X 0,Y 434.722,Z 900.047,A -85,B 0,C 180,E1 12986.824,E2 12986.824} C_VEL
LIN {X 0,Y 440.214,Z 877.863,A -85,B 0,C 180,E1 12986.146,E2 12986.146} C_VEL
LIN {X 0,Y 444.672,Z 856.323,A -85,B 0,C 180,E1 12985.614,E2 12985.614} C_VEL
LIN {X 0,Y 448.675,Z 831.952,A -85,B 0,C 180,E1 12985.135,E2 12985.135} C_VEL
LIN {X 0,Y 452.432,Z 795.842,A -85,B 0,C 180,E1 12984.549,E2 12984.549} C_VEL
LIN {X 0,Y 471.356,Z 581.094,A -85,B 0,C 180,E1 12981.291,E2 12981.291} C_VEL
LIN {X 0,Y 466.234,Z 572.138,A -85,B 0,C 180,E1 12978.636,E2 12978.636} C_VEL
LIN {X 0,Y 461.788,Z 564.441,A -85,B 0,C 180,E1 12975.832,E2 12975.832} C_VEL
LIN {X 0,Y 459.275,Z 560.381,A -85,B 0,C 180,E1 12973.92,E2 12973.92} C_VEL
LIN {X 0,Y 456.85,Z 556.264,A -85,B 0,C 180,E1 12971.616,E2 12971.616} C_VEL
LIN {X 0,Y 454.586,Z 552.032,A -85,B 0,C 180,E1 12968.475,E2 12968.475} C_VEL
LIN {X 0,Y 453.136,Z 550.65,A -85,B 0,C 180,E1 12964.175,E2 12964.175} C_VEL
LIN {X 0,Y 453.816,Z 551.335,A -85,B 0,C 180,E1 12960.126,E2 12960.126} C_VEL
LIN {X 0,Y 454.588,Z 552.099,A -85,B 0,C 180,E1 12958.614,E2 12958.614} C_VEL
LIN {X 0,Y 456.859,Z 556.25,A -85,B 0,C 180,E1 12955.481,E2 12955.481} C_VEL
LIN {X 0,Y 460.28,Z 561.934,A -85,B 0,C 180,E1 12952.385,E2 12952.385} C_VEL
LIN {X 0,Y 463.384,Z 567.313,A -85,B 0,C 180,E1 12950.185,E2 12950.185} C_VEL
LIN {X 0,Y 467.105,Z 573.602,A -85,B 0,C 180,E1 12947.985,E2 12947.985} C_VEL
LIN {X 0,Y 471.4,Z 581.446,A -85,B 0,C 180,E1 12945.778,E2 12945.778} C_VEL
LIN {X 0,Y 451.949,Z 802.57,A -85,B 0,C 180,E1 12942.421,E2 12942.421} C_VEL
LIN {X 0,Y 448.209,Z 837.225,A -85,B 0,C 180,E1 12941.849,E2 12941.849} C_VEL
LIN {X 0,Y 444.34,Z 860.465,A -85,B 0,C 180,E1 12941.394,E2 12941.394} C_VEL
LIN {X 0,Y 439.872,Z 881.795,A -85,B 0,C 180,E1 12940.878,E2 12940.878} C_VEL
LIN {X 0,Y 434.394,Z 903.728,A -85,B 0,C 180,E1 12940.223,E2 12940.223} C_VEL
LIN {X 0,Y 426.227,Z 931.218,A -85,B 0,C 180,E1 12939.198,E2 12939.198} C_VEL
LIN {X 0,Y 418.389,Z 953.661,A -85,B 0,C 180,E1 12938.16,E2 12938.16} C_VEL
LIN {X 0,Y 410.619,Z 973.582,A -85,B 0,C 180,E1 12937.069,E2 12937.069} C_VEL
LIN {X 0,Y 402.25,Z 993.095,A -85,B 0,C 180,E1 12935.816,E2 12935.816} C_VEL
LIN {X 0,Y 391.717,Z 1015.544,A -85,B 0,C 180,E1 12934.12,E2 12934.12} C_VEL
LIN {X 0,Y 380.495,Z 1036.982,A -85,B 0,C 180,E1 12932.159,E2 12932.159} C_VEL
LIN {X 0,Y 370.702,Z 1054.412,A -85,B 0,C 180,E1 12930.284,E2 12930.284} C_VEL
LIN {X 0,Y 360.999,Z 1070.714,A -85,B 0,C 180,E1 12928.244,E2 12928.244} C_VEL
LIN {X 0,Y 350.264,Z 1087.873,A -85,B 0,C 180,E1 12925.731,E2 12925.731} C_VEL
LIN {X 0,Y 337.449,Z 1107.285,A -85,B 0,C 180,E1 12922.29,E2 12922.29} C_VEL
LIN {X 0,Y 328.039,Z 1121.015,A -85,B 0,C 180,E1 12919.371,E2 12919.371} C_VEL
LIN {X 0,Y 319.422,Z 1133.359,A -85,B 0,C 180,E1 12916.309,E2 12916.309} C_VEL
LIN {X 0,Y 311.204,Z 1145.107,A -85,B 0,C 180,E1 12912.898,E2 12912.898} C_VEL
LIN {X 0,Y 301.974,Z 1158.514,A -85,B 0,C 180,E1 12908.255,E2 12908.255} C_VEL
LIN {X 0,Y 294.716,Z 1169.394,A -85,B 0,C 180,E1 12903.573,E2 12903.573} C_VEL
LIN {X 0,Y 289.887,Z 1177.215,A -85,B 0,C 180,E1 12899.553,E2 12899.553} C_VEL
LIN {X 0,Y 286.137,Z 1183.919,A -85,B 0,C 180,E1 12895.455,E2 12895.455} C_VEL
LIN {X 0,Y 283.285,Z 1189.815,A -85,B 0,C 180,E1 12891.101,E2 12891.101} C_VEL
LIN {X 0,Y 281.254,Z 1195.221,A -85,B 0,C 180,E1 12886.098,E2 12886.098} C_VEL
LIN {X 0,Y 280.208,Z 1199.392,A -85,B 0,C 180,E1 12880.693,E2 12880.693} C_VEL
LIN {X 0,Y 279.95,Z 1201.656,A -85,B 0,C 180,E1 12876.151,E2 12876.151} C_VEL
LIN {X 0,Y 279.914,Z 1202.753,A -85,B 0,C 180,E1 12872.047,E2 12872.047} C_VEL
LIN {X 0,Y 279.913,Z 1202.928,A -85,B 0,C 180,E1 12867.953,E2 12867.953} C_VEL
LIN {X 0,Y 279.949,Z 1202.188,A -85,B 0,C 180,E1 12863.849,E2 12863.849} C_VEL
LIN {X 0,Y 280.198,Z 1200.426,A -85,B 0,C 180,E1 12859.514,E2 12859.514} C_VEL
LIN {X 0,Y 280.956,Z 1197.663,A -85,B 0,C 180,E1 12855.153,E2 12855.153} C_VEL
LIN {X 0,Y 282.465,Z 1193.889,A -85,B 0,C 180,E1 12850.78,E2 12850.78} C_VEL
LIN {X 0,Y 284.952,Z 1189.083,A -85,B 0,C 180,E1 12846.421,E2 12846.421} C_VEL
LIN {X 0,Y 288.551,Z 1183.184,A -85,B 0,C 180,E1 12842.084,E2 12842.084} C_VEL
LIN {X 0,Y 293.802,Z 1175.554,A -85,B 0,C 180,E1 12837.473,E2 12837.473} C_VEL
LIN {X 0,Y 302.508,Z 1163.961,A -85,B 0,C 180,E1 12831.876,E2 12831.876} C_VEL
LIN {X 0,Y 310.413,Z 1153.894,A -85,B 0,C 180,E1 12827.935,E2 12827.935} C_VEL
LIN {X 0,Y 319.291,Z 1142.838,A -85,B 0,C 180,E1 12824.295,E2 12824.295} C_VEL
LIN {X 0,Y 329.205,Z 1130.487,A -85,B 0,C 180,E1 12820.865,E2 12820.865} C_VEL
LIN {X 0,Y 342.714,Z 1113.26,A -85,B 0,C 180,E1 12816.929,E2 12816.929} C_VEL
LIN {X 0,Y 353.946,Z 1098.365,A -85,B 0,C 180,E1 12814.138,E2 12814.138} C_VEL
LIN {X 0,Y 364.656,Z 1083.611,A -85,B 0,C 180,E1 12811.789,E2 12811.789} C_VEL
LIN {X 0,Y 375.25,Z 1068.293,A -85,B 0,C 180,E1 12809.7,E2 12809.7} C_VEL
LIN {X 0,Y 387.023,Z 1050.287,A -85,B 0,C 180,E1 12807.61,E2 12807.61} C_VEL
LIN {X 0,Y 400.75,Z 1027.45,A -85,B 0,C 180,E1 12805.421,E2 12805.421} C_VEL
LIN {X 0,Y 411.208,Z 1008.424,A -85,B 0,C 180,E1 12803.901,E2 12803.901} C_VEL
LIN {X 0,Y 420.804,Z 989.495,A -85,B 0,C 180,E1 12802.617,E2 12802.617} C_VEL
LIN {X 0,Y 429.811,Z 970.022,A -85,B 0,C 180,E1 12801.486,E2 12801.486} C_VEL
LIN {X 0,Y 440.209,Z 944.924,A -85,B 0,C 180,E1 12800.273,E2 12800.273} C_VEL
LIN {X 0,Y 448.736,Z 920.816,A -85,B 0,C 180,E1 12799.331,E2 12799.331} C_VEL
LIN {X 0,Y 455.124,Z 900.135,A -85,B 0,C 180,E1 12798.665,E2 12798.665} C_VEL
LIN {X 0,Y 460.657,Z 879.278,A -85,B 0,C 180,E1 12798.108,E2 12798.108} C_VEL
LIN {X 0,Y 465.65,Z 856.727,A -85,B 0,C 180,E1 12797.624,E2 12797.624} C_VEL
LIN {X 0,Y 470.564,Z 826.915,A -85,B 0,C 180,E1 12797.106,E2 12797.106} C_VEL
LIN {X 0,Y 476.209,Z 772.22,A -85,B 0,C 180,E1 12796.284,E2 12796.284} C_VEL
LIN {X 0,Y 493.745,Z 596.413,A -85,B 0,C 180,E1 12793.706,E2 12793.706} C_VEL
LIN {X 0,Y 492.007,Z 593.156,A -85,B 0,C 180,E1 12792.261,E2 12792.261} C_VEL
LIN {X 0,Y 490.216,Z 589.823,A -85,B 0,C 180,E1 12790.459,E2 12790.459} C_VEL
LIN {X 0,Y 488.326,Z 586.033,A -85,B 0,C 180,E1 12787.767,E2 12787.767} C_VEL
LIN {X 0,Y 487.071,Z 584.431,A -85,B 0,C 180,E1 12783.531,E2 12783.531} C_VEL
LIN {X 0,Y 487.662,Z 585.395,A -85,B 0,C 180,E1 12780.352,E2 12780.352} C_VEL
LIN {X 0,Y 488.57,Z 586.503,A -85,B 0,C 180,E1 12778.593,E2 12778.593} C_VEL
LIN {X 0,Y 491.055,Z 591.33,A -85,B 0,C 180,E1 12775.445,E2 12775.445} C_VEL
LIN {X 0,Y 493.396,Z 595.688,A -85,B 0,C 180,E1 12773.367,E2 12773.367} C_VEL
LIN {X 0,Y 493.679,Z 596.451,A -85,B 0,C 180,E1 12773.127,E2 12773.127} C_VEL
LIN {X 0,Y 471.794,Z 815.379,A -85,B 0,C 180,E1 12769.908,E2 12769.908} C_VEL
LIN {X 0,Y 468.663,Z 838.183,A -85,B 0,C 180,E1 12769.537,E2 12769.537} C_VEL
LIN {X 0,Y 464.593,Z 860.116,A -85,B 0,C 180,E1 12769.123,E2 12769.123} C_VEL
LIN {X 0,Y 459.122,Z 883.768,A -85,B 0,C 180,E1 12768.564,E2 12768.564} C_VEL
LIN {X 0,Y 451.239,Z 911.207,A -85,B 0,C 180,E1 12767.733,E2 12767.733} C_VEL
LIN {X 0,Y 443.942,Z 932.679,A -85,B 0,C 180,E1 12766.927,E2 12766.927} C_VEL
LIN {X 0,Y 436.322,Z 952.514,A -85,B 0,C 180,E1 12766.042,E2 12766.042} C_VEL
LIN {X 0,Y 427.972,Z 971.984,A -85,B 0,C 180,E1 12765.026,E2 12765.026} C_VEL
LIN {X 0,Y 416.943,Z 995.237,A -85,B 0,C 180,E1 12763.582,E2 12763.582} C_VEL
LIN {X 0,Y 404.791,Z 1017.853,A -85,B 0,C 180,E1 12761.866,E2 12761.866} C_VEL
LIN {X 0,Y 394.649,Z 1035.245,A -85,B 0,C 180,E1 12760.307,E2 12760.307} C_VEL
LIN {X 0,Y 384.064,Z 1052.149,A -85,B 0,C 180,E1 12758.544,E2 12758.544} C_VEL
LIN {X 0,Y 372.573,Z 1069.391,A -85,B 0,C 180,E1 12756.429,E2 12756.429} C_VEL
LIN {X 0,Y 357.913,Z 1089.908,A -85,B 0,C 180,E1 12753.373,E2 12753.373} C_VEL
LIN {X 0,Y 347.072,Z 1104.229,A -85,B 0,C 180,E1 12750.796,E2 12750.796} C_VEL
LIN {X 0,Y 336.953,Z 1117.149,A -85,B 0,C 180,E1 12748.066,E2 12748.066} C_VEL
LIN {X 0,Y 327.068,Z 1129.451,A -85,B 0,C 180,E1 12745.013,E2 12745.013} C_VEL
LIN {X 0,Y 316.069,Z 1143.054,A -85,B 0,C 180,E1 12740.983,E2 12740.983} C_VEL
LIN {X 0,Y 305.8,Z 1155.556,A -85,B 0,C 180,E1 12736.376,E2 12736.376} C_VEL
LIN {X 0,Y 298.466,Z 1164.799,A -85,B 0,C 180,E1 12732.236,E2 12732.236} C_VEL
LIN {X 0,Y 292.497,Z 1172.729,A -85,B 0,C 180,E1 12727.974,E2 12727.974} C_VEL
LIN {X 0,Y 287.021,Z 1180.797,A -85,B 0,C 180,E1 12722.68,E2 12722.68} C_VEL
LIN {X 0,Y 283.21,Z 1187.207,A -85,B 0,C 180,E1 12717.092,E2 12717.092} C_VEL
LIN {X 0,Y 281.36,Z 1191.189,A -85,B 0,C 180,E1 12712.569,E2 12712.569} C_VEL
LIN {X 0,Y 280.412,Z 1193.979,A -85,B 0,C 180,E1 12708.287,E2 12708.287} C_VEL
LIN {X 0,Y 280.036,Z 1195.748,A -85,B 0,C 180,E1 12704.262,E2 12704.262} C_VEL
LIN {X 0,Y 279.931,Z 1196.679,A -85,B 0,C 180,E1 12700.288,E2 12700.288} C_VEL
LIN {X 0,Y 279.92,Z 1196.789,A -85,B 0,C 180,E1 12696.357,E2 12696.357} C_VEL
LIN {X 0,Y 279.935,Z 1196.091,A -85,B 0,C 180,E1 12692.457,E2 12692.457} C_VEL
LIN {X 0,Y 280.099,Z 1194.482,A -85,B 0,C 180,E1 12688.364,E2 12688.364} C_VEL
LIN {X 0,Y 280.623,Z 1191.827,A -85,B 0,C 180,E1 12684.069,E2 12684.069} C_VEL
LIN {X 0,Y 281.778,Z 1188.179,A -85,B 0,C 180,E1 12679.781,E2 12679.781} C_VEL
LIN {X 0,Y 283.749,Z 1183.518,A -85,B 0,C 180,E1 12675.512,E2 12675.512} C_VEL
LIN {X 0,Y 286.671,Z 1177.816,A -85,B 0,C 180,E1 12671.284,E2 12671.284} C_VEL
LIN {X 0,Y 290.859,Z 1170.688,A -85,B 0,C 180,E1 12666.928,E2 12666.928} C_VEL
LIN {X 0,Y 297.394,Z 1160.723,A -85,B 0,C 180,E1 12661.921,E2 12661.921} C_VEL
LIN {X 0,Y 305.281,Z 1149.165,A -85,B 0,C 180,E1 12657.289,E2 12657.289} C_VEL
LIN {X 0,Y 312.736,Z 1138.636,A -85,B 0,C 180,E1 12653.739,E2 12653.739} C_VEL
LIN {X 0,Y 320.717,Z 1127.428,A -85,B 0,C 180,E1 12650.507,E2 12650.507} C_VEL
LIN {X 0,Y 330.529,Z 1113.566,A -85,B 0,C 180,E1 12647.107,E2 12647.107} C_VEL
LIN {X 0,Y 342.907,Z 1095.437,A -85,B 0,C 180,E1 12643.445,E2 12643.445} C_VEL
LIN {X 0,Y 352.973,Z 1080.072,A -85,B 0,C 180,E1 12640.859,E2 12640.859} C_VEL
LIN {X 0,Y 362.759,Z 1064.468,A -85,B 0,C 180,E1 12638.611,E2 12638.611} C_VEL
LIN {X 0,Y 373.674,Z 1046.104,A -85,B 0,C 180,E1 12636.351,E2 12636.351} C_VEL
LIN {X 0,Y 386.081,Z 1023.402,A -85,B 0,C 180,E1 12634.033,E2 12634.033} C_VEL
LIN {X 0,Y 395.596,Z 1004.475,A -85,B 0,C 180,E1 12632.417,E2 12632.417} C_VEL
LIN {X 0,Y 403.96,Z 986.419,A -85,B 0,C 180,E1 12631.086,E2 12631.086} C_VEL
LIN {X 0,Y 412.515,Z 966.22,A -85,B 0,C 180,E1 12629.805,E2 12629.805} C_VEL
LIN {X 0,Y 422.016,Z 941.159,A -85,B 0,C 180,E1 12628.48,E2 12628.48} C_VEL
LIN {X 0,Y 427.024,Z 926.273,A -85,B 0,C 180,E1 12627.813,E2 12627.813} C_VEL
LIN {X 0,Y 428.872,Z 919.379,A -85,B 0,C 180,E1 12627.402,E2 12627.402} C_VEL
LIN {X 0,Y 431.459,Z 902.27,A -85,B 0,C 180,E1 12626.033,E2 12626.033} C_VEL
LIN {X 0,Y 432.97,Z 895.159,A -85,B 0,C 180,E1 12625.678,E2 12625.678} C_VEL
LIN {X 0,Y 438.614,Z 871.976,A -85,B 0,C 180,E1 12625.014,E2 12625.014} C_VEL
LIN {X 0,Y 444.204,Z 842.681,A -85,B 0,C 180,E1 12624.369,E2 12624.369} C_VEL
LIN {X 0,Y 447.384,Z 819.316,A -85,B 0,C 180,E1 12623.961,E2 12623.961} C_VEL
LIN {X 0,Y 465.781,Z 616.347,A -85,B 0,C 180,E1 12620.883,E2 12620.883} C_VEL
LIN {X 0,Y 468.501,Z 586.539,A -85,B 0,C 180,E1 12620.43,E2 12620.43} C_VEL
LIN {X 0,Y 463.893,Z 578.274,A -85,B 0,C 180,E1 12617.888,E2 12617.888} C_VEL
LIN {X 0,Y 459.948,Z 571.342,A -85,B 0,C 180,E1 12615.251,E2 12615.251} C_VEL
LIN {X 0,Y 458.051,Z 568.16,A -85,B 0,C 180,E1 12613.744,E2 12613.744} C_VEL
LIN {X 0,Y 455.642,Z 564.017,A -85,B 0,C 180,E1 12611.391,E2 12611.391} C_VEL
LIN {X 0,Y 453.338,Z 559.611,A -85,B 0,C 180,E1 12607.987,E2 12607.987} C_VEL
LIN {X 0,Y 452.148,Z 558.565,A -85,B 0,C 180,E1 12603.169,E2 12603.169} C_VEL
LIN {X 0,Y 453.503,Z 559.887,A -85,B 0,C 180,E1 12598.8,E2 12598.8} C_VEL
LIN {X 0,Y 455.755,Z 564.121,A -85,B 0,C 180,E1 12595.596,E2 12595.596} C_VEL
LIN {X 0,Y 459.039,Z 569.758,A -85,B 0,C 180,E1 12592.553,E2 12592.553} C_VEL
LIN {X 0,Y 462.186,Z 575.311,A -85,B 0,C 180,E1 12590.285,E2 12590.285} C_VEL
LIN {X 0,Y 466.129,Z 582.244,A -85,B 0,C 180,E1 12587.928,E2 12587.928} C_VEL
LIN {X 0,Y 468.563,Z 586.824,A -85,B 0,C 180,E1 12586.634,E2 12586.634} C_VEL
LIN {X 0,Y 448.743,Z 807.452,A -85,B 0,C 180,E1 12583.304,E2 12583.304} C_VEL
LIN {X 0,Y 445.257,Z 837.847,A -85,B 0,C 180,E1 12582.8,E2 12582.8} C_VEL
LIN {X 0,Y 441.375,Z 860.695,A -85,B 0,C 180,E1 12582.356,E2 12582.356} C_VEL
LIN {X 0,Y 436.791,Z 882.168,A -85,B 0,C 180,E1 12581.843,E2 12581.843} C_VEL
LIN {X 0,Y 431.005,Z 904.853,A -85,B 0,C 180,E1 12581.171,E2 12581.171} C_VEL
LIN {X 0,Y 422.564,Z 932.443,A -85,B 0,C 180,E1 12580.144,E2 12580.144} C_VEL
LIN {X 0,Y 414.855,Z 954.059,A -85,B 0,C 180,E1 12579.152,E2 12579.152} C_VEL
LIN {X 0,Y 406.896,Z 974.044,A -85,B 0,C 180,E1 12578.067,E2 12578.067} C_VEL
LIN {X 0,Y 398.158,Z 993.961,A -85,B 0,C 180,E1 12576.795,E2 12576.795} C_VEL
LIN {X 0,Y 386.692,Z 1017.628,A -85,B 0,C 180,E1 12574.995,E2 12574.995} C_VEL
LIN {X 0,Y 375.947,Z 1037.608,A -85,B 0,C 180,E1 12573.162,E2 12573.162} C_VEL
LIN {X 0,Y 365.929,Z 1054.981,A -85,B 0,C 180,E1 12571.294,E2 12571.294} C_VEL
LIN {X 0,Y 355.664,Z 1071.744,A -85,B 0,C 180,E1 12569.185,E2 12569.185} C_VEL
LIN {X 0,Y 343.456,Z 1090.698,A -85,B 0,C 180,E1 12566.366,E2 12566.366} C_VEL
LIN {X 0,Y 331.774,Z 1107.658,A -85,B 0,C 180,E1 12563.286,E2 12563.286} C_VEL
LIN {X 0,Y 322.065,Z 1121.346,A -85,B 0,C 180,E1 12560.346,E2 12560.346} C_VEL
LIN {X 0,Y 313.155,Z 1133.653,A -85,B 0,C 180,E1 12557.253,E2 12557.253} C_VEL
LIN {X 0,Y 304.274,Z 1145.878,A -85,B 0,C 180,E1 12553.635,E2 12553.635} C_VEL
LIN {X 0,Y 293.999,Z 1160.116,A -85,B 0,C 180,E1 12548.489,E2 12548.489} C_VEL
LIN {X 0,Y 287.462,Z 1169.556,A -85,B 0,C 180,E1 12544.296,E2 12544.296} C_VEL
LIN {X 0,Y 282.402,Z 1177.347,A -85,B 0,C 180,E1 12540.182,E2 12540.182} C_VEL
LIN {X 0,Y 278.296,Z 1184.33,A -85,B 0,C 180,E1 12535.768,E2 12535.768} C_VEL
LIN {X 0,Y 274.909,Z 1191.188,A -85,B 0,C 180,E1 12530.436,E2 12530.436} C_VEL
LIN {X 0,Y 272.911,Z 1196.495,A -85,B 0,C 180,E1 12524.86,E2 12524.86} C_VEL
LIN {X 0,Y 272.175,Z 1199.61,A -85,B 0,C 180,E1 12520.37,E2 12520.37} C_VEL
LIN {X 0,Y 271.949,Z 1201.612,A -85,B 0,C 180,E1 12516.121,E2 12516.121} C_VEL
LIN {X 0,Y 271.915,Z 1202.657,A -85,B 0,C 180,E1 12512.107,E2 12512.107} C_VEL
LIN {X 0,Y 271.913,Z 1202.848,A -85,B 0,C 180,E1 12507.893,E2 12507.893} C_VEL
LIN {X 0,Y 271.953,Z 1202.125,A -85,B 0,C 180,E1 12503.668,E2 12503.668} C_VEL
LIN {X 0,Y 272.23,Z 1200.378,A -85,B 0,C 180,E1 12499.204,E2 12499.204} C_VEL
LIN {X 0,Y 273.064,Z 1197.632,A -85,B 0,C 180,E1 12494.714,E2 12494.714} C_VEL
LIN {X 0,Y 274.702,Z 1193.877,A -85,B 0,C 180,E1 12490.214,E2 12490.214} C_VEL
LIN {X 0,Y 277.368,Z 1189.09,A -85,B 0,C 180,E1 12485.736,E2 12485.736} C_VEL
LIN {X 0,Y 281.395,Z 1182.942,A -85,B 0,C 180,E1 12481.103,E2 12481.103} C_VEL
LIN {X 0,Y 287.341,Z 1174.901,A -85,B 0,C 180,E1 12476.169,E2 12476.169} C_VEL
LIN {X 0,Y 296.026,Z 1163.958,A -85,B 0,C 180,E1 12470.831,E2 12470.831} C_VEL
LIN {X 0,Y 304.674,Z 1153.504,A -85,B 0,C 180,E1 12466.695,E2 12466.695} C_VEL
LIN {X 0,Y 313.712,Z 1142.738,A -85,B 0,C 180,E1 12463.125,E2 12463.125} C_VEL
LIN {X 0,Y 323.876,Z 1130.571,A -85,B 0,C 180,E1 12459.722,E2 12459.722} C_VEL
LIN {X 0,Y 337.775,Z 1113.495,A -85,B 0,C 180,E1 12455.799,E2 12455.799} C_VEL
LIN {X 0,Y 349.924,Z 1097.885,A -85,B 0,C 180,E1 12452.882,E2 12452.882} C_VEL
LIN {X 0,Y 361.034,Z 1083.005,A -85,B 0,C 180,E1 12450.538,E2 12450.538} C_VEL
LIN {X 0,Y 371.944,Z 1067.642,A -85,B 0,C 180,E1 12448.474,E2 12448.474} C_VEL
LIN {X 0,Y 384.763,Z 1048.494,A -85,B 0,C 180,E1 12446.295,E2 12446.295} C_VEL
LIN {X 0,Y 398.086,Z 1026.624,A -85,B 0,C 180,E1 12444.254,E2 12444.254} C_VEL
LIN {X 0,Y 408.388,Z 1008.253,A -85,B 0,C 180,E1 12442.812,E2 12442.812} C_VEL
LIN {X 0,Y 418.168,Z 989.317,A -85,B 0,C 180,E1 12441.548,E2 12441.548} C_VEL
LIN {X 0,Y 427.747,Z 968.948,A -85,B 0,C 180,E1 12440.392,E2 12440.392} C_VEL
LIN {X 0,Y 438.709,Z 942.565,A -85,B 0,C 180,E1 12439.16,E2 12439.16} C_VEL
LIN {X 0,Y 446.589,Z 920.592,A -85,B 0,C 180,E1 12438.327,E2 12438.327} C_VEL
LIN {X 0,Y 453.074,Z 899.892,A -85,B 0,C 180,E1 12437.675,E2 12437.675} C_VEL
LIN {X 0,Y 458.716,Z 878.897,A -85,B 0,C 180,E1 12437.127,E2 12437.127} C_VEL
LIN {X 0,Y 463.892,Z 855.759,A -85,B 0,C 180,E1 12436.645,E2 12436.645} C_VEL
LIN {X 0,Y 468.836,Z 825.637,A -85,B 0,C 180,E1 12436.133,E2 12436.133} C_VEL
LIN {X 0,Y 475.622,Z 760.408,A -85,B 0,C 180,E1 12435.166,E2 12435.166} C_VEL
LIN {X 0,Y 491.699,Z 602.533,A -85,B 0,C 180,E1 12432.872,E2 12432.872} C_VEL
LIN {X 0,Y 489.134,Z 597.712,A -85,B 0,C 180,E1 12430.363,E2 12430.363} C_VEL
LIN {X 0,Y 487.284,Z 593.934,A -85,B 0,C 180,E1 12427.665,E2 12427.665} C_VEL
LIN {X 0,Y 486.094,Z 592.354,A -85,B 0,C 180,E1 12423.42,E2 12423.42} C_VEL
LIN {X 0,Y 486.884,Z 593.596,A -85,B 0,C 180,E1 12419.882,E2 12419.882} C_VEL
LIN {X 0,Y 487.512,Z 594.388,A -85,B 0,C 180,E1 12418.707,E2 12418.707} C_VEL
LIN {X 0,Y 489.886,Z 599.126,A -85,B 0,C 180,E1 12415.61,E2 12415.61} C_VEL
LIN {X 0,Y 491.644,Z 602.526,A -85,B 0,C 180,E1 12413.96,E2 12413.96} C_VEL
LIN {X 0,Y 469.756,Z 816.94,A -85,B 0,C 180,E1 12410.836,E2 12410.836} C_VEL
LIN {X 0,Y 466.586,Z 839.284,A -85,B 0,C 180,E1 12410.475,E2 12410.475} C_VEL
LIN {X 0,Y 462.295,Z 861.8,A -85,B 0,C 180,E1 12410.054,E2 12410.054} C_VEL
LIN {X 0,Y 455.936,Z 888.314,A -85,B 0,C 180,E1 12409.42,E2 12409.42} C_VEL
LIN {X 0,Y 448.441,Z 913.195,A -85,B 0,C 180,E1 12408.66,E2 12408.66} C_VEL
LIN {X 0,Y 441.255,Z 933.844,A -85,B 0,C 180,E1 12407.891,E2 12407.891} C_VEL
LIN {X 0,Y 433.513,Z 953.55,A -85,B 0,C 180,E1 12407.022,E2 12407.022} C_VEL
LIN {X 0,Y 424.521,Z 974.034,A -85,B 0,C 180,E1 12405.96,E2 12405.96} C_VEL
LIN {X 0,Y 412.031,Z 999.302,A -85,B 0,C 180,E1 12404.373,E2 12404.373} C_VEL
LIN {X 0,Y 401.408,Z 1018.567,A -85,B 0,C 180,E1 12402.906,E2 12402.906} C_VEL
LIN {X 0,Y 390.985,Z 1036.009,A -85,B 0,C 180,E1 12401.357,E2 12401.357} C_VEL
LIN {X 0,Y 380.243,Z 1052.739,A -85,B 0,C 180,E1 12399.623,E2 12399.623} C_VEL
LIN {X 0,Y 367.73,Z 1071.011,A -85,B 0,C 180,E1 12397.383,E2 12397.383} C_VEL
LIN {X 0,Y 353.417,Z 1090.366,A -85,B 0,C 180,E1 12394.487,E2 12394.487} C_VEL
LIN {X 0,Y 341.622,Z 1105.441,A -85,B 0,C 180,E1 12391.759,E2 12391.759} C_VEL
LIN {X 0,Y 330.683,Z 1118.911,A -85,B 0,C 180,E1 12388.865,E2 12388.865} C_VEL
LIN {X 0,Y 318.378,Z 1133.72,A -85,B 0,C 180,E1 12385.051,E2 12385.051} C_VEL
LIN {X 0,Y 307.013,Z 1146.908,A -85,B 0,C 180,E1 12380.814,E2 12380.814} C_VEL
LIN {X 0,Y 298.44,Z 1156.958,A -85,B 0,C 180,E1 12376.916,E2 12376.916} C_VEL
LIN {X 0,Y 291.144,Z 1165.737,A -85,B 0,C 180,E1 12372.842,E2 12372.842} C_VEL
LIN {X 0,Y 284.077,Z 1174.763,A -85,B 0,C 180,E1 12367.765,E2 12367.765} C_VEL
LIN {X 0,Y 278.421,Z 1182.616,A -85,B 0,C 180,E1 12362.054,E2 12362.054} C_VEL
LIN {X 0,Y 275.376,Z 1187.588,A -85,B 0,C 180,E1 12357.46,E2 12357.46} C_VEL
LIN {X 0,Y 273.497,Z 1191.34,A -85,B 0,C 180,E1 12353.027,E2 12353.027} C_VEL
LIN {X 0,Y 272.46,Z 1194.112,A -85,B 0,C 180,E1 12348.619,E2 12348.619} C_VEL
LIN {X 0,Y 272.051,Z 1195.863,A -85,B 0,C 180,E1 12344.473,E2 12344.473} C_VEL
LIN {X 0,Y 271.935,Z 1196.754,A -85,B 0,C 180,E1 12340.594,E2 12340.594} C_VEL
LIN {X 0,Y 271.919,Z 1196.891,A -85,B 0,C 180,E1 12336.545,E2 12336.545} C_VEL
LIN {X 0,Y 271.937,Z 1196.152,A -85,B 0,C 180,E1 12332.318,E2 12332.318} C_VEL
LIN {X 0,Y 272.118,Z 1194.526,A -85,B 0,C 180,E1 12328.105,E2 12328.105} C_VEL
LIN {X 0,Y 272.695,Z 1191.854,A -85,B 0,C 180,E1 12323.685,E2 12323.685} C_VEL
LIN {X 0,Y 273.953,Z 1188.19,A -85,B 0,C 180,E1 12319.273,E2 12319.273} C_VEL
LIN {X 0,Y 276.076,Z 1183.511,A -85,B 0,C 180,E1 12314.885,E2 12314.885} C_VEL
LIN {X 0,Y 279.195,Z 1177.79,A -85,B 0,C 180,E1 12310.546,E2 12310.546} C_VEL
LIN {X 0,Y 283.649,Z 1170.643,A -85,B 0,C 180,E1 12306.086,E2 12306.086} C_VEL
LIN {X 0,Y 290.842,Z 1160.189,A -85,B 0,C 180,E1 12300.78,E2 12300.78} C_VEL
